	441:
		tmrA_10.PT := T#60S;
		tmrA_10.IN := TRUE;
		stepA := stepA + 1;
			 
	442:// 到達中間感應器，停止
		IF NOT io.i202 OR tmrA_10.q THEN
			io.q201 := FALSE;
			tmrA_10.in := FALSE;
					  
			IF NOT io.i202 THEN
				stepA := stepA + 1;
			ELSIF tmrA_10.q THEN
				stepA := stepA + 10000;
			END_IF
		END_IF
			 
	443:
		tmrA_1.PT := T#500ms;
		tmrA_1.IN := TRUE;
		IF tmrA_1.Q THEN
			tmrA_1.IN := FALSE;
			io.q202 := TRUE;
			IF io.i202 THEN
				// 如果上升到超過感應器，下降到有之後，繼續下降到脫離
				stepA := 444;
			ELSE
				// 停在感應器上，下降到脫離
				stepA := 445;
			END_IF
		END_IF
			
	444:// 
		IF NOT io.i202 THEN
			stepA := stepA + 1;
		END_IF
				  
	445:
		IF io.i202 THEN
			io.q202 := FALSE;
			stepA := stepA + 1;
		END_IF
				  
	446:
		CarLift_WaitSync.0 := TRUE;
		stepA := 450;
				  
//	450: // 等待主油壓切至慢速模式 ，完成後由主流程跳步
				  
	451: // 用慢速上升
		io.q201 := TRUE;
		IF NOT io.i202 THEN
			io.q201 := FALSE;
			stepA := stepA + 1;
		END_IF
				  
	452: // 用慢速上升
		io.q201 := TRUE;
		IF NOT io.i202 THEN
			io.q201 := FALSE;
			stepA := stepA + 1;
		END_IF
		
	453:
		stepA := 0;
	{endregion}
			  
	{region "============= 位置不確定  ============="}	
	470: // 位置不確定(沒在任何感應器上) ，先下降
		io.q201 := FALSE;
		io.q202 := TRUE;
		stepA := stepA + 1;
			 
	471:
		tmrA_10.PT := T#60S;
		tmrA_10.IN := TRUE;
		stepA := stepA + 1;
			 
	472:// 通過中間感應器 或 到達下方感應器
		IF NOT io.i202 OR NOT io.i203 OR tmrA_10.q THEN
			tmrA_10.in := FALSE;
					  
			IF NOT io.i203 THEN
				// 到達下方感應器
				io.q202 := FALSE;
				stepA := 440;
			ELSIF NOT io.i202 THEN
				// 通過中間感應器
				stepA := 480;
			ELSIF tmrA_10.q THEN
				stepA := stepA + 10000;
			END_IF
		END_IF
			 
	480: 
		IF io.i202 THEN
			io.q202 := FALSE;
			stepA := stepA + 1;
		END_IF
			
	481:// 
		CarLift_WaitSync.0 := TRUE;
		stepA := 420;
	{endregion}
		
END_CASE
{endregion}

{region "============= 台車B中位移動  ============="}
CASE stepB OF
	400: // 判斷位置
		IF NOT io.i205 THEN
			stepB := 0;
		ELSE
			IF NOT io.i204 THEN
				// 位置在上限
				stepB := 410;
			ELSIF NOT io.i206 THEN
				// 位置在下限
				stepB := 440;
			ELSE
			    // 位置不確定
				stepB := 470;
		 	END_IF
		END_IF
	{region "============= 位置在上限  ============="}	
	410: // 位置在上限，下降
		io.q203 := FALSE;
		io.q204 := TRUE;
		stepB := stepB + 1;
			 
	411:
		tmrB_10.PT := T#60S;
		tmrB_10.IN := TRUE;
		stepB := stepB + 1;
			 
	412://
		IF NOT io.i205 OR tmrB_10.q THEN
			tmrB_10.in := FALSE;
			IF NOT io.i205 THEN
				stepB := stepB + 1;
			ELSIF tmrB_10.q THEN
				stepB := stepB + 10000;
			END_IF
		END_IF
			 
	413: // 先降過頭在慢速升回
		IF io.i205 THEN
			io.q204 := FALSE;
			stepB := stepB + 1;
		END_IF
				  
	414:
		CarLift_WaitSync.1 := TRUE;
		stepB := 420;
				  
//	420: // 等待主油壓切至慢速模式 ，完成後由主流程跳步
		
				  
	421: // 用慢速上升
		io.q203 := TRUE;
		IF NOT io.i205 THEN
			io.q203 := FALSE;
			stepB := stepB + 1;
		END_IF
				  
	422: // 用慢速上升
		io.q203 := TRUE;
		IF NOT io.i205 THEN
			io.q203 := FALSE;
			stepB := stepB + 1;
		END_IF
		
	423:
		stepB := 0;
	{endregion}
	{region "============= 位置在下限  ============="}	
	440: // 位置在下限，上升
		io.q203 := TRUE;
		io.q204 := FALSE;
		stepB := stepB + 1;
			 
	441:
		tmrB_10.PT := T#60S;
		tmrB_10.IN := TRUE;
		stepB := stepB + 1;
			 
	442:// 到達中間感應器，停止
		IF NOT io.i205 OR tmrB_10.q THEN
			io.q203 := FALSE;
			tmrB_10.in := FALSE;
					  
			IF NOT io.i205 THEN
				stepB := stepB + 1;
			ELSIF tmrB_10.q THEN
				stepB := stepB + 10000;
			END_IF
		END_IF
			 
	443:
		tmrB_1.PT := T#500ms;
		tmrB_1.IN := TRUE;
		IF tmrB_1.Q THEN
			tmrB_1.IN := FALSE;
			io.q204 := TRUE;
			IF io.i205 THEN
				// 如果上升到超過感應器，下降到有之後，繼續下降到脫離
				stepB := 444;
			ELSE
				// 停在感應器上，下降到脫離
				stepB := 445;
			END_IF
		END_IF
			
	444:// 
		IF NOT io.i205 THEN
			stepB := stepB + 1;
		END_IF
				  
	445:
		IF io.i205 THEN
			io.q204 := FALSE;
			stepB := stepB + 1;
		END_IF
				  
	446:
		CarLift_WaitSync.1 := TRUE;
		stepB := 450;
				  
//	450: // 等待主油壓切至慢速模式 ，完成後由主流程跳步
				  
	451: // 用慢速上升
		io.q203 := TRUE;
		IF NOT io.i205 THEN
			io.q203 := FALSE;
			stepB := stepB + 1;
		END_IF
				  
	452: // 用慢速上升
		io.q203 := TRUE;
		IF NOT io.i205 THEN
			io.q203 := FALSE;
			stepB := stepB + 1;
		END_IF
		
	453:
		stepB := 0;
	{endregion}
			  
	{region "============= 位置不確定  ============="}	
	470: // 位置不確定(沒在任何感應器上) ，先下降
		io.q203 := FALSE;
		io.q204 := TRUE;
		stepB := stepB + 1;
			 
	471:
		tmrB_10.PT := T#60S;
		tmrB_10.IN := TRUE;
		stepB := stepB + 1;
			 
	472:// 通過中間感應器 或 到達下方感應器
		IF NOT io.i205 OR NOT io.i206 OR tmrB_10.q THEN
			tmrB_10.in := FALSE;
					  
			IF NOT io.i206 THEN
				// 到達下方感應器
				io.q204 := FALSE;
				stepB := 440;
			ELSIF NOT io.i205 THEN
				// 通過中間感應器
				stepB := 480;
			ELSIF tmrB_10.q THEN
				stepB := stepB + 10000;
			END_IF
		END_IF
			 
	480: 
		IF io.i205 THEN
			io.q204 := FALSE;
			stepB := stepB + 1;
		END_IF
			
	481:// 
		CarLift_WaitSync.1 := TRUE;
		stepB := 420;
	{endregion}
		
END_CASE
{endregion}
	 
{region "============= 台車C中位移動  ============="}
CASE stepC OF
	400: // 判斷位置
		IF NOT io.i208 THEN
			stepC := 0;
		ELSE
			IF NOT io.i207 THEN
				// 位置在上限
				stepC := 410;
			ELSIF NOT io.i209 THEN
				// 位置在下限
				stepC := 440;
			ELSE
			    // 位置不確定
				stepC := 470;
		 	END_IF
		END_IF
	{region "============= 位置在上限  ============="}	
	410: // 位置在上限，下降
		io.q205 := FALSE;
		io.q206 := TRUE;
		stepC := stepC + 1;
			 
	411:
		tmrC_10.PT := T#60S;
		tmrC_10.IN := TRUE;
		stepC := stepC + 1;
			 
	412://
		IF NOT io.i208 OR tmrC_10.q THEN
			tmrC_10.in := FALSE;
			IF NOT io.i208 THEN
				stepC := stepC + 1;
			ELSIF tmrC_10.q THEN
				stepC := stepC + 10000;
			END_IF
		END_IF
			 
	413: // 先降過頭在慢速升回
		IF io.i208 THEN
			io.q206 := FALSE;
			stepC := stepC + 1;
		END_IF
				  
	414:
		CarLift_WaitSync.2 := TRUE;
		stepC := 420;
				  
//	420: // 等待主油壓切至慢速模式 ，完成後由主流程跳步
		
				  
	421: // 用慢速上升
		io.q205 := TRUE;
		IF NOT io.i208 THEN
			io.q205 := FALSE;
			stepC := stepC + 1;
		END_IF
				  
	422: // 用慢速上升
		io.q205 := TRUE;
		IF NOT io.i208 THEN
			io.q205 := FALSE;
			stepC := stepC + 1;
		END_IF
		
	423:
		stepC := 0;
	{endregion}
	{region "============= 位置在下限  ============="}	
	440: // 位置在下限，上升
		io.q205 := TRUE;
		io.q206 := FALSE;
		stepC := stepC + 1;
			 
	441:
		tmrC_10.PT := T#60S;
		tmrC_10.IN := TRUE;
		stepC := stepC + 1;
			 
	442:// 到達中間感應器，停止
		IF NOT io.i208 OR tmrC_10.q THEN
			io.q205 := FALSE;
			tmrC_10.in := FALSE;
					  
			IF NOT io.i208 THEN
				stepC := stepC + 1;
			ELSIF tmrC_10.q THEN
				stepC := stepC + 10000;
			END_IF
		END_IF
			 
	443:
		tmrC_1.PT := T#500ms;
		tmrC_1.IN := TRUE;
		IF tmrC_1.Q THEN
			tmrC_1.IN := FALSE;
			io.q206 := TRUE;
			IF io.i208 THEN
				// 如果上升到超過感應器，下降到有之後，繼續下降到脫離
				stepC := 444;
			ELSE
				// 停在感應器上，下降到脫離
				stepC := 445;
			END_IF
		END_IF
			
	444:// 
		IF NOT io.i208 THEN
			stepC := stepC + 1;
		END_IF
				  
	445:
		IF io.i208 THEN
			io.q206 := FALSE;
			stepC := stepC + 1;
		END_IF
				  
	446:
		CarLift_WaitSync.2 := TRUE;
		stepC := 450;
				  
//	450: // 等待主油壓切至慢速模式 ，完成後由主流程跳步
				  
	451: // 用慢速上升
		io.q205 := TRUE;
		IF NOT io.i208 THEN
			io.q205 := FALSE;
			stepC := stepC + 1;
		END_IF
				  
	452: // 用慢速上升
		io.q205 := TRUE;
		IF NOT io.i208 THEN
			io.q205 := FALSE;
			stepC := stepC + 1;
		END_IF
		
	453:
		stepC := 0;
	{endregion}
			  
	{region "============= 位置不確定  ============="}	
	470: // 位置不確定(沒在任何感應器上) ，先下降
		io.q205 := FALSE;
		io.q206 := TRUE;
		stepC := stepC + 1;
			 
	471:
		tmrC_10.PT := T#60S;
		tmrC_10.IN := TRUE;
		stepC := stepC + 1;
			 
	472:// 通過中間感應器 或 到達下方感應器
		IF NOT io.i208 OR NOT io.i209 OR tmrC_10.q THEN
			tmrC_10.in := FALSE;
					  
			IF NOT io.i209 THEN
				// 到達下方感應器
				io.q206 := FALSE;
				stepC := 440;
			ELSIF NOT io.i208 THEN
				// 通過中間感應器
				stepC := 480;
			ELSIF tmrC_10.q THEN
				stepC := stepC + 10000;
			END_IF
		END_IF
			 
	480: 
		IF io.i208 THEN
			io.q206 := FALSE;
			stepC := stepC + 1;
		END_IF
			
	481:// 
		CarLift_WaitSync.2 := TRUE;
		stepC := 420;
	{endregion}
		
END_CASE
{endregion}
	 
{region "============= 台車D中位移動  ============="}
CASE stepD OF
	400: // 判斷位置
		IF NOT io.i211 THEN
			stepD := 0;
		ELSE
			IF NOT io.i210 THEN
				// 位置在上限
				stepD := 410;
			ELSIF NOT io.i212 THEN
				// 位置在下限
				stepD := 440;
			ELSE
			    // 位置不確定
				stepD := 470;
		 	END_IF
		END_IF
	{region "============= 位置在上限  ============="}	
	410: // 位置在上限，下降
		io.q207 := FALSE;
		io.q208 := TRUE;
		stepD := stepD + 1;
			 
	411:
		tmrD_10.PT := T#60S;
		tmrD_10.IN := TRUE;
		stepD := stepD + 1;
			 
	412://
		IF NOT io.i211 OR tmrD_10.q THEN
			tmrD_10.in := FALSE;
			IF NOT io.i211 THEN
				stepD := stepD + 1;
			ELSIF tmrD_10.q THEN
				stepD := stepD + 10000;
			END_IF
		END_IF
			 
	413: // 先降過頭在慢速升回
		IF io.i211 THEN
			io.q208 := FALSE;
			stepD := stepD + 1;
		END_IF
				  
	414:
		CarLift_WaitSync.3 := TRUE;
		stepD := 420;
				  
//	420: // 等待主油壓切至慢速模式 ，完成後由主流程跳步
		
				  
	421: // 用慢速上升
		io.q207 := TRUE;
		IF NOT io.i211 THEN
			io.q207 := FALSE;
			stepD := stepD + 1;
		END_IF
				  
	422: // 用慢速上升
		io.q207 := TRUE;
		IF NOT io.i211 THEN
			io.q207 := FALSE;
			stepD := stepD + 1;
		END_IF
		
	423:
		stepD := 0;
	{endregion}
	{region "============= 位置在下限  ============="}	
	440: // 位置在下限，上升
		io.q207 := TRUE;
		io.q208 := FALSE;
		stepD := stepD + 1;
			 
	441:
		tmrD_10.PT := T#60S;
		tmrD_10.IN := TRUE;
		stepD := stepD + 1;
			 
	442:// 到達中間感應器，停止
		IF NOT io.i211 OR tmrD_10.q THEN
			io.q207 := FALSE;
			tmrD_10.in := FALSE;
					  
			IF NOT io.i211 THEN
				stepD := stepD + 1;
			ELSIF tmrD_10.q THEN
				stepD := stepD + 10000;
			END_IF
		END_IF
			 
	443:
		tmrD_1.PT := T#500ms;
		tmrD_1.IN := TRUE;
		IF tmrD_1.Q THEN
			tmrD_1.IN := FALSE;
			io.q208 := TRUE;
			IF io.i211 THEN
				// 如果上升到超過感應器，下降到有之後，繼續下降到脫離
				stepD := 444;
			ELSE
				// 停在感應器上，下降到脫離
				stepD := 445;
			END_IF
		END_IF
			
	444:// 
		IF NOT io.i211 THEN
			stepD := stepD + 1;
		END_IF
				  
	445:
		IF io.i211 THEN
			io.q208 := FALSE;
			stepD := stepD + 1;
		END_IF
				  
	446:
		CarLift_WaitSync.3 := TRUE;
		stepD := 450;
				  
//	450: // 等待主油壓切至慢速模式 ，完成後由主流程跳步
				  
	451: // 用慢速上升
		io.q207 := TRUE;
		IF NOT io.i211 THEN
			io.q207 := FALSE;
			stepD := stepD + 1;
		END_IF
				  
	452: // 用慢速上升
		io.q207 := TRUE;
		IF NOT io.i211 THEN
			io.q207 := FALSE;
			stepD := stepD + 1;
		END_IF
		
	453:
		stepD := 0;
	{endregion}
			  
	{region "============= 位置不確定  ============="}	
	470: // 位置不確定(沒在任何感應器上) ，先下降
		io.q207 := FALSE;
		io.q208 := TRUE;
		stepD := stepD + 1;
			 
	471:
		tmrD_10.PT := T#60S;
		tmrD_10.IN := TRUE;
		stepD := stepD + 1;
			 
	472:// 通過中間感應器 或 到達下方感應器
		IF NOT io.i211 OR NOT io.i212 OR tmrD_10.q THEN
			tmrD_10.in := FALSE;
					  
			IF NOT io.i212 THEN
				// 到達下方感應器
				io.q208 := FALSE;
				stepD := 440;
			ELSIF NOT io.i211 THEN
				// 通過中間感應器
				stepD := 480;
			ELSIF tmrD_10.q THEN
				stepD := stepD + 10000;
			END_IF
		END_IF
			 
	480: 
		IF io.i211 THEN
			io.q208 := FALSE;
			stepD := stepD + 1;
		END_IF
			
	481:// 
		CarLift_WaitSync.3 := TRUE;
		stepD := 420;
	{endregion}
		
END_CASE
{endregion}
END_ACTION

ACTION step_6_CarLift_Down:
CASE step OF
	600:
		IF (CarLift_Select AND 16#F) = 0 THEN
			CarLift_Select := 15;
		END_IF
		step := step + 1;
	
	601:
		io.q301 := TRUE;
		IF CarLift_Select.0 THEN
			stepA := 600;
		END_IF
		
		IF CarLift_Select.1 THEN
			stepB := 600;
		END_IF
		
		IF CarLift_Select.2 THEN
			stepC := 600;
		END_IF
		
		IF CarLift_Select.3 THEN
			stepD := 600;
		END_IF
		
		step := step + 1;
		
	602:
		IF stepA = 0 AND stepB = 0 AND stepC = 0 AND stepD = 0 THEN
			step := step + 1;
		ELSIF stepA > 10000 OR stepB > 10000 OR stepC > 10000 OR stepD > 10000 THEN
			step := step + 10000;
		END_IF
		
	603:
		io.q301 := FALSE;
		CarLift_Select := 0;
		bDone := TRUE;
		step := 0;
		
END_CASE

{region "============= 台車A下降  ============="}
CASE stepA OF
	600: // 啟動上升
		io.q201 := FALSE;
		io.q202 := TRUE;
		stepA := stepA + 1;
		
	601: // 啟動超時計時器
		tmrA_10.PT := T#20S;
		tmrA_10.IN := TRUE;
		stepA := stepA + 1;
		
	602: // 等待
		IF NOT io.i203 OR tmrA_10.q THEN
			tmrA_10.in := FALSE;
			
			IF NOT io.i203 THEN
				stepA := stepA + 1;
			ELSIF tmrA_10.q THEN
				io.q202 := FALSE;
				stepA := stepA + 10000;
			END_IF
		END_IF
		
	603: // 成功之後等待1秒
		tmrA_1.PT := T#1S;
		tmrA_1.IN := TRUE;
		IF tmrA_1.Q THEN
			tmrA_1.IN := FALSE;
			io.q202 := FALSE;
			stepA := stepA + 1;
		END_IF
		
	604:
		stepA := 0;
		
END_CASE
{endregion}

{region "============= 台車B下降  ============="}
CASE stepB OF
	600: // 啟動上升
		io.q203 := FALSE;
		io.q204 := TRUE;
		stepB := stepB + 1;
		
	601: // 啟動超時計時器
		tmrB_10.PT := T#20S;
		tmrB_10.IN := TRUE;
		stepB := stepB + 1;
		
	602: // 等待
		IF NOT io.i206 OR tmrB_10.q THEN
			tmrB_10.in := FALSE;
			
			IF NOT io.i206 THEN
				stepB := stepB + 1;
			ELSIF tmrB_10.q THEN
				io.q204 := FALSE;
				stepB := stepB + 10000;
			END_IF
		END_IF
		
	603: // 成功之後等待1秒
		tmrB_1.PT := T#1S;
		tmrB_1.IN := TRUE;
		IF tmrB_1.Q THEN
			io.q204 := FALSE;
			stepB := stepB + 1;
		END_IF
		
	604:
		stepB := 0;
		
END_CASE
{endregion}

{region "============= 台車C下降  ============="}
CASE stepC OF
	600: // 啟動上升
		io.q205 := FALSE;
		io.q206 := TRUE;
		stepC := stepC + 1;
		
	601: // 啟動超時計時器
		tmrC_10.PT := T#20S;
		tmrC_10.IN := TRUE;
		stepC := stepC + 1;
		
	602: // 等待
		IF NOT io.i209 OR tmrC_10.q THEN
			tmrC_10.in := FALSE;
			
			IF NOT io.i209 THEN
				stepC := stepC + 1;
			ELSIF tmrC_10.q THEN
				io.q206 := FALSE;
				stepC := stepC + 10000;
			END_IF
		END_IF
		
	603: // 成功之後等待1秒
		tmrC_1.PT := T#1S;
		tmrC_1.IN := TRUE;
		IF tmrC_1.Q THEN
			io.q206 := FALSE;
			stepC := stepC + 1;
		END_IF
		
	604:
		stepC := 0;
		
END_CASE
{endregion}

{region "============= 台車D下降  ============="}
CASE stepD OF
	600: // 啟動上升
		io.q207 := FALSE;
		io.q208 := TRUE;
		stepD := stepD + 1;
		
	601: // 啟動超時計時器
		tmrD_10.PT := T#20S;
		tmrD_10.IN := TRUE;
		stepD := stepD + 1;
		
	602: // 等待
		IF NOT io.i212 OR tmrD_10.q THEN
			tmrD_10.in := FALSE;
			
			IF NOT io.i212 THEN
				stepD := stepD + 1;
			ELSIF tmrD_10.q THEN
				io.q207 := FALSE;
				stepD := stepD + 10000;
			END_IF
		END_IF
		
	603: // 成功之後等待1秒
		tmrD_1.PT := T#1S;
		tmrD_1.IN := TRUE;
		IF tmrD_1.Q THEN
			io.q208 := FALSE;
			stepD := stepD + 1;
		END_IF
		
	604:
		stepD := 0;
		
END_CASE
{endregion}
END_ACTION

ACTION step1_1_Pull_over:
CASE step1 OF
	100:// 檢查
		TryCount := 0;
		step1 := step1 + 1;
		
	101:
		step1 := 110;
		
	110: // 啟動靠邊油壓閥
		io.q302 := TRUE;
		IF NOT bbuzy THEN
			io.q301 := TRUE;
		END_IF
		step1 := step1 + 1;
		
	111: // 確定原點已脫離
		IF io.i401 THEN
			step1 := step1 + 1;
		END_IF
		
	112: // 程序暫停5秒
		tmr1_01.PT := T#4S;
		tmr1_01.IN := io.i402 OR io.i404;
		
		tmr1_02.PT := T#5S;
		tmr1_02.IN := TRUE;
		IF tmr1_01.Q OR tmr1_02.q THEN
			tmr1_01.IN := FALSE;
			tmr1_02.IN := FALSE;
			
			IF tmr1_01.q THEN
				step1 := 190;
			ELSIF tmr1_02.Q THEN
				step1 := step1 + 1;
			END_IF
		END_IF
		
	113:
		step1 := 120;
		
	120:// 沒推到待命位置
		io.q302 := FALSE;
		step1 := step1 + 1;
		
	121: // 等待回原點
		tmr01.PT := T#1S;
		tmr01.IN := (NOT io.i401 AND NOT io.i403 AND NOT io.i405 AND NOT io.i407);
		IF tmr01.Q THEN
			tmr01.IN := FALSE;
			step1 := step1 + 1;
		END_IF
		
	122: 
		
		IF TryCount < 4 THEN
			TryCount := TryCount + 1;
			step1 := 110;
		ELSE
			TryCount := 0;
			step1 := step1 + 10000;
		END_IF
		
		
	190:
		
		tmr1_01.PT := T#3S;
		tmr1_01.IN := TRUE;
		IF tmr1_01.Q THEN
			tmr1_01.IN := FALSE;
			step1 := step1 + 1;
		END_IF
		
	191:
		io.q302 := FALSE;
		bdone1 := TRUE;
		step1 := 0;
END_CASE
END_ACTION

ACTION step1_2_Pull_over_Jog:
CASE step1 OF
	200:// 檢查
		step1 := step1 + 1;
		
	201:
		IF io.q302 THEN
			step1 := 220;
		ELSE
			step1 := 210;
		END_IF
		
		
	210: // 啟動靠邊油壓閥
		io.q302 := TRUE;
		IF NOT bbuzy THEN
			io.q301 := TRUE;
		END_IF
		step1 := step1 + 1;
		
	211: // 確定原點已脫離
		tmr01.PT := T#4S;
		tmr01.IN := (io.i401 AND io.i403 AND io.i405 AND io.i407);
		IF tmr01.Q THEN
			tmr01.IN := FALSE;
			step1 := step1 + 1;
		END_IF
		
	212:
		step1 := 290;
		
	220: // 關閉靠邊油壓閥
		io.q302 := FALSE;
		IF NOT bbuzy THEN
			io.q301 := TRUE;
		END_IF
		step1 := step1 + 1;
		
	221: // 等待回原點
		tmr01.PT := T#4S;
		tmr01.IN := (NOT io.i401 AND NOT io.i403 AND NOT io.i405 AND NOT io.i407);
		IF tmr01.Q THEN
			tmr01.IN := FALSE;
			step1 := step1 + 1;
		END_IF
		
	222: 
		step1 := 290;
		
		
	290:
		bdone1 := TRUE;
		io.q301 := FALSE;
		step1 := 0;
END_CASE
END_ACTION

METHOD Stop : BOOL
VAR_INPUT
END_VAR
step := 100;
END_METHOD

ACTION tmrAct:
tmr01();

tmr1_01();
tmr1_02();

tmrA_1();
tmrA_10();
tmrB_1();
tmrB_10();
tmrC_1();
tmrC_10();
tmrD_1();
tmrD_10();


tmr_pump();
END_ACTION

END_PROGRAM

// ---- POUs/動作流程控制/滾輪整料/PullOver.TcPOU
PROGRAM PullOver
VAR
	step: UINT;
	
	
END_VAR

VAR_OUTPUT
	bBuzy: BOOL;
	bError: BOOL;
	bDone: BOOL;
	iErrorId : DINT;
END_VAR

IF (EStop OR SystemError OR Input.Feed_Reset) AND bBuzy THEN
	IF bBuzy THEN
		step := step  + 10000;
	END_IF
END_IF

bBuzy := (step >= 1 AND step < 10000);
bError := (step > 10000);


CASE step OF
	1:
		bDone := FALSE;
		step := 10;	
(*	=====================================
				測高不再原點
	=====================================*)
	10:
		IF HeightMeasurer.at_Home THEN
			step := 100;
		ELSE
			step := step + 1;
		END_IF
		
	11:
		HeightMeasurer.Homing();
		step := step + 1;
		
	12:
		IF HeightMeasurer.bBuzy OR HeightMeasurer.bError THEN
			step := step + 1;
		END_IF
		
	13:
		IF HeightMeasurer.bDone THEN
			step := step + 1;
		ELSIF HeightMeasurer.bError THEN
			step := step + 10000;
		END_IF
		
	14:
		step := 100;
		
		
(*	=====================================
				靠邊啟動
	=====================================*)
	100:
		Hydraulic.Over_Pull(0);
		step := step + 1;
		
	101:
		IF (Hydraulic.bBuzy1 OR Hydraulic.bError1) THEN
			step := step + 1;
		END_IF
		
	102:
		IF Hydraulic.bDone1 THEN
			step := step + 1;
		ELSIF Hydraulic.bError1 THEN
			step := step + 10000;
		END_IF
		
	103:
		step := 110;
		
(*	=====================================
				高度測量
	=====================================*)
	110:
		HeightMeasurer.Measure();
		step := step + 1;
		
	111:
		IF (HeightMeasurer.bBuzy OR HeightMeasurer.bError) THEN
			step := step + 1;
		END_IF
		
	112:
		IF HeightMeasurer.bDone THEN
			step := step + 1;
		ELSIF HeightMeasurer.bError THEN
			step := step + 10000;
		END_IF
		
	113:
		step := 120;
		
	
	120:
		bDone := TRUE;
		step := 0;
END_CASE

IF Input.PullOver_Start AND NOT bBuzy THEN
	step := 1;
END_IF

Output.PullOver_bBuzy := bBuzy;
Output.PullOver_bDone := bDone;
Output.PullOver_bError := bError;

METHOD Start
VAR_INPUT
END_VAR
step := 1;
END_METHOD

END_PROGRAM

// ---- POUs/硬體控制/進料滾輪/FeedRoller.TcPOU
PROGRAM FeedRoller
VAR
	step: INT;
	
	_run : BOOL;
	
	start_RTrig : R_TRIG;
	start_FTrig : F_TRIG;
	
	_bError : BOOL;
	
	tmr0 : TON;
	tmr1 : TON;
END_VAR

VAR_OUTPUT
	bDone: BOOL;
	bBuzy: BOOL;
	bError: BOOL;
	
	Move_Fwd : BOOL;
	Move_Rev : BOOL;
	At_Up : BOOL;
	At_Down : BOOL;
END_VAR

// 沒 SystemError 是避免進料機影響到整體動作
IF (EStop OR Input.Feed_Reset) AND bBuzy THEN
	IF bBuzy THEN
		step := step  + 10000;
	END_IF
	IO.q102 := FALSE;
	IO.q103 := FALSE;
	IO.q309 := FALSE;
	IO.q310 := FALSE;
	IO.q311 := FALSE;
	IO.q312 := FALSE;
END_IF


// 外部 送入 啟動訊號
start_RTrig(CLK := Input.In_Moter_Start );

IF	start_RTrig.q THEN
	step := 1;
END_IF

// 外部 解除 啟動訊號
start_FTrig(CLK := Input.In_Moter_Start);

IF start_FTrig.Q THEN
	step := 100;
END_IF

// 執行動作發生錯誤
_bError := step > 10000;

IF _bError THEN
	_run := FALSE;
	IO.q103 := FALSE;
	IO.q102 := FALSE;
END_IF

// 馬達 動作中過載檢知
IF IO.i109 AND step > 0 AND step < 10000 THEN
	step := 10900;
END_IF

bBuzy := step > 0 AND step < 10000;
bError := step > 10000;

IF bBuzy THEN
	bDone := FALSE;
END_IF

step_0_Auto_Start();
step_1_Auto_Stop();
step_7_Jog_FwdRev();
step_8_Jog_UpDown();

Output.In_Moter_Running := step > 0 OR Move_Fwd OR Move_Rev;
Output.In_Moter_Error := _bError;

tmr0();
tmr1();

Move_Fwd	:= IO.q103;
Move_Rev	:= IO.q102;
At_Up		:= IO.i411;
At_Down		:= IO.i412;

METHOD Jog_Down
VAR_INPUT
END_VAR
bDone := FALSE;

step := 820;
END_METHOD

METHOD Jog_Fwd
VAR_INPUT
END_VAR
bDone := FALSE;

step := 700;
END_METHOD

METHOD Jog_Rev
VAR_INPUT
END_VAR
bDone := FALSE;

step := 720;
END_METHOD

METHOD Jog_Stop
VAR_INPUT
END_VAR
step := 780;
END_METHOD

METHOD Jog_Up
VAR_INPUT
END_VAR
bDone := FALSE;

step := 800;
END_METHOD

ACTION step_0_Auto_Start:
CASE step OF
	1:
		IF IO.i109 THEN
			// 滾輪馬達保護氣跳脫
			step := step + 10000;
// 		ELSIF NOT IO.i314 THEN
// 			// 測高位置錯誤
// 			step := step + 10000;
		ELSE
			step := step + 1;
		END_IF
		
	2:
		IF HeightMeasurer.bBuzy THEN
			// 測高動作執行中
			step := step + 10000;
		ELSE
			// 進料動作執行中
			step := step + 1;
		END_IF
		
	3:
		step := 10;
		
	10:
		IO.q309 := TRUE;
		IO.q310 := FALSE;
		IO.q311 := TRUE;
		IO.q312 := FALSE;
		tmr1.PT := T#10S;
		tmr1.IN := TRUE;
		step := step + 1;
		
	11:
		IF NOT IO.i412 OR tmr1.Q THEN
			IO.q309 := FALSE;
			IO.q311 := FALSE;
			tmr1.IN := FALSE;
			IF NOT IO.i412 THEN
				step := step + 1;
			ELSE
				// 上升超時
				step := step + 10000;
			END_IF
		END_IF
		
	12:
		step := 20;
		
	20:
		IO.q103 := TRUE;
		_run :=	TRUE;
		step := 0;
END_CASE
END_ACTION

ACTION step_1_Auto_Stop:
CASE step OF
	100:
		IO.q309 := FALSE;
		IO.q311 := FALSE;
		IO.q103 := FALSE;
		step := step + 1;
		
	101:
		tmr0.PT:= T#1S;
		tmr0.IN := TRUE;
		IF tmr0.Q THEN
			tmr0.IN := FALSE;
			step := step + 1;
		END_IF
		
	102:
		step := 110;
		
	110:
		IO.q310 := TRUE;
		IO.q312 := TRUE;
		tmr1.PT := T#10S;
		tmr1.IN := TRUE;
		step := step + 1;
		
	111:
		IF IO.i412 OR tmr1.Q THEN
			IO.q310 := FALSE;
			IO.q312 := FALSE;
			tmr1.IN := FALSE;
			IF IO.i412 THEN
				step := step + 1;
			ELSE
				// 上升超時
				step := step + 10000;
			END_IF
		END_IF
		
	112:
		_run :=	FALSE;
		step := 0;
END_CASE
END_ACTION

ACTION step_7_Jog_FwdRev:
CASE step OF
	700:
		IO.q102 := FALSE;
		IF IO.i109 THEN
			// 滾輪馬達保護氣跳脫
			step := step + 10000;
// 		ELSIF NOT IO.i314 THEN
// 			// 測高位置錯誤
// 			step := step + 10000;
		ELSE
			step := step + 1;
		END_IF
		
	701: // 啟動馬達
		IO.q103 := TRUE;
		bDone := TRUE;
		step := 0;
		
	
		


	720:
		IO.q103 := FALSE;
		IF IO.i109 THEN
			// 滾輪馬達保護氣跳脫
			step := step + 10000;
// 		ELSIF NOT IO.i314 THEN
// 			// 測高位置錯誤
// 			step := step + 10000;
		ELSE
			step := step + 1;
		END_IF
		
	721:
		IO.q102 := TRUE;
		bDone := TRUE;
		step := 0;
		
	
		


	780:
		IO.q102 := FALSE;
		IO.q103 := FALSE;
		bDone := TRUE;
		step := 0;
END_CASE
END_ACTION

ACTION step_8_Jog_UpDown:
CASE step OF
	800:
		IO.q309 := TRUE;
		IO.q310 := FALSE;
		IO.q311 := TRUE;
		IO.q312 := FALSE;
		
		tmr1.PT := T#10S;
		tmr1.IN := TRUE;
		step := step + 1;
		
	801: // 滾輪上升
		IF NOT IO.i412 OR tmr1.Q THEN
			IO.q309 := FALSE;
			IO.q311 := FALSE;
			tmr1.IN := FALSE;
			IF NOT IO.i412 THEN
				step := step + 1;
			ELSE
				// 上升超時
				step := step + 10000;
			END_IF
		END_IF
		
	802:
		bDone := TRUE;
		step := 0;
		
	
		


	820:
		IO.q309 := FALSE;
		IO.q310 := TRUE;
		IO.q311 := FALSE;
		IO.q312 := TRUE;
		
		tmr1.PT := T#10S;
		tmr1.IN := TRUE;
		step := step + 1;
		
	821: // 滾輪上升
		IF IO.i412 OR tmr1.Q THEN
			IO.q310 := FALSE;
			IO.q312 := FALSE;
			tmr1.IN := FALSE;
			IF IO.i412 THEN
				step := step + 1;
			ELSE
				// 上升超時
				step := step + 10000;
			END_IF
		END_IF
		
	822:
		bDone := TRUE;
		step := 0;
		
	

END_CASE
END_ACTION

END_PROGRAM

// ---- POUs/硬體控制/出料滾輪/ProductRoller.TcPOU
PROGRAM ProductRoller
VAR
	step: INT;
	
	_run : BOOL;
	
	start_RTrig : R_TRIG;
	start_FTrig : F_TRIG;
	
	_bError : BOOL;
	
	
	tmr0 : TON;
	tmr1 : TON;
	
	Roller_Up :BOOL;
	Roller_Down :BOOL;
	
	Roller_Fwd :BOOL;
	Roller_Rev :BOOL;
END_VAR

VAR_OUTPUT
	bDone: BOOL;
	bBuzy: BOOL;
	bError: BOOL;
	
	Move_Fwd : BOOL;
	Move_Rev : BOOL;
	At_Up : BOOL;
	At_Down : BOOL;
END_VAR


// 沒 SystemError 是避免進料機影響到整體動作
IF (EStop OR Input.Feed_Reset) AND bBuzy THEN
	IF bBuzy THEN
		step := step  + 10000;
	END_IF
	IO.q114 := FALSE;
	IO.q115 := FALSE;
	IO.q305 := FALSE;
	IO.q306 := FALSE;
END_IF


// 外部 送入 啟動訊號
start_RTrig(CLK := Input.Out_Moter_Start);

IF	start_RTrig.q THEN
	step := 1;
END_IF

// 外部 解除 啟動訊號
start_FTrig(CLK := Input.Out_Moter_Start);

IF start_FTrig.Q THEN
	step := 100;
END_IF



// 執行動作發生錯誤
_bError := step > 10000;

IF _bError THEN
	_run := FALSE;
	IO.q114 := FALSE;
	IO.q115 := FALSE;
END_IF

// 馬達 動作中過載檢知
IF IO.i109 AND step > 0 AND step < 10000 THEN
	step := 10900;
END_IF

bBuzy := step > 0 AND step < 10000;
bError := step > 10000;

IF bBuzy THEN
	bDone := FALSE;
END_IF

IF NOT Pause THEN
	step_0_Auto_Start();
	step_1_Auto_Stop();

	IO.q115 := Roller_Fwd;
	IO.q114 := Roller_Rev;
	IO.q306 := Roller_Up;
	IO.q305 := Roller_Down;
ELSE
	IO.q115 := FALSE;
	IO.q114 := FALSE;
	IO.q306 := FALSE;
	IO.q305 := FALSE;
END_IF

step_7_Jog_FwdRev();
step_8_Jog_UpDown();



Output.Out_Moter_Running := step > 0 OR Move_Fwd OR Move_Rev;;
Output.Out_Moter_Error := _bError;

tmr0();
tmr1();

Move_Fwd	:= IO.q115;
Move_Rev	:= IO.q114;
At_Up		:= IO.i316;
At_Down		:= IO.i315;

METHOD Jog_Down
VAR_INPUT
END_VAR
bDone := FALSE;

step := 820;
END_METHOD

METHOD Jog_Fwd
VAR_INPUT
END_VAR
bDone := FALSE;

step := 700;
END_METHOD

METHOD Jog_Rev
VAR_INPUT
END_VAR
bDone := FALSE;

step := 720;
END_METHOD

METHOD Jog_Stop
VAR_INPUT
END_VAR
step := 780;
END_METHOD

METHOD Jog_Up
VAR_INPUT
END_VAR
bDone := FALSE;

step := 800;
END_METHOD

ACTION step_0_Auto_Start:
CASE step OF
	1:
		IF IO.i112 THEN
			// 滾輪馬達保護氣跳脫
			step := step + 10000;
// 		ELSIF IO.i113 THEN
// 			
		ELSE
			step := step + 1;
		END_IF
		
	2:
		step := 10;
		
	10:
		Roller_Down := FALSE;
		Roller_Up 	:= TRUE;
		tmr1.PT := T#10S;
		tmr1.IN := TRUE;
		step := step + 1;
		
	11:
		IF NOT IO.i315 OR tmr1.Q THEN
			Roller_Up := FALSE;
			tmr1.IN := FALSE;
			IF NOT IO.i315 THEN
				step := step + 1;
			ELSE
				// 上升超時
				step := step + 10000;
			END_IF
		END_IF
		
	12:
		step := 20;
		
	20:
		Roller_Rev := FALSE;
		Roller_Fwd := TRUE;
		_run :=	TRUE;
		step := 0;
END_CASE
END_ACTION

ACTION step_1_Auto_Stop:
CASE step OF
	100:
		Roller_Rev := FALSE;
		Roller_Fwd := FALSE;
		step := step + 1;
		
	101:
		tmr0.PT:= T#1S;
		tmr0.IN := TRUE;
		IF tmr0.Q THEN
			tmr0.IN := FALSE;
			step := step + 1;
		END_IF
		
	102:
		step := 110;
		
	110:
		Roller_Down := TRUE;
		Roller_Up := FALSE;
		tmr1.PT := T#10S;
		tmr1.IN := TRUE;
		step := step + 1;
		
	111:
		IF IO.i315 OR tmr1.Q THEN
			Roller_Down := FALSE;
			tmr1.IN := FALSE;
			IF IO.i315 THEN
				step := step + 1;
			ELSE
				// 上升超時
				step := step + 10000;
			END_IF
		END_IF
		
	112:
		_run :=	FALSE;
		step := 0;
END_CASE
END_ACTION

ACTION step_7_Jog_FwdRev:
CASE step OF
	700:
		Roller_Rev := FALSE;
		IF IO.i112 THEN
			// 滾輪馬達保護氣跳脫
			step := step + 10000;
		ELSE
			step := step + 1;
		END_IF
		
	701: // 啟動馬達
		Roller_Fwd := TRUE;
		bDone := TRUE;
		step := 0;
		
	
		


	720:
		Roller_Fwd := FALSE;
		IF IO.i112 THEN
			// 滾輪馬達保護氣跳脫
			step := step + 10000;
		ELSE
			step := step + 1;
		END_IF
		
	721:
		Roller_Rev := TRUE;
		bDone := TRUE;
		step := 0;
		
	
		


	780:
		Roller_Rev := FALSE;
		Roller_Fwd := FALSE;
		bDone := TRUE;
		step := 0;
END_CASE
END_ACTION

ACTION step_8_Jog_UpDown:
CASE step OF
	800:
		Roller_Up 	:= TRUE;
		Roller_Down := FALSE;
		
		tmr1.PT := T#10S;
		tmr1.IN := TRUE;
		step := step + 1;
		
	801: // 滾輪上升
		IF NOT IO.i315 OR tmr1.Q THEN
			Roller_Up := FALSE;
			tmr1.IN := FALSE;
			IF not IO.i315 THEN
				step := step + 1;
			ELSE
				// 上升超時
				step := step + 10000;
			END_IF
		END_IF
		
	802:
		bDone := TRUE;
		step := 0;
		
	
		


	820:
		Roller_Up := FALSE;
		Roller_Down := TRUE;
		
		tmr1.PT := T#10S;
		tmr1.IN := TRUE;
		step := step + 1;
		
	821: // 滾輪上升
		IF IO.i315 OR tmr1.Q THEN
			Roller_Down := FALSE;
			tmr1.IN := FALSE;
			IF IO.i315 THEN
				step := step + 1;
			ELSE
				// 上升超時
				step := step + 10000;
			END_IF
		END_IF
		
	822:
		bDone := TRUE;
		step := 0;
		
	

END_CASE
END_ACTION

END_PROGRAM

// ---- POUs/資料轉換/HMI_WEB_dataConver.TcPOU
PROGRAM HMI_WEB_dataConver
VAR
END_VAR

Hmi_Web.Car_pos := Axis.FeedCar.Pos;

END_PROGRAM

// ---- POUs/硬體控制/台車/編碼器/MM540.TcPOU
FUNCTION_BLOCK MM540
VAR_INPUT
END_VAR
VAR_OUTPUT
	// 等待觸發中
	bActive : BOOL;
	// 忙碌中
	bBuzy : BOOL;
	// 已完成
	bDone : BOOL;
	// 發生錯誤
	bError : BOOL;
END_VAR
VAR
	FeedCar_Enc_raw : MM540_Raw;
	
	Step : INT;
	
	_SetPos : DINT;
	
	_timeout	: TIME := T#10S;
	
	_timeTmr	: TON;
END_VAR

bBuzy := Step > 0 AND Step < 10000;
bActive := FeedCar_Enc_raw.Inc_Preload_Trigger > 0 AND bBuzy;
bError := Step >= 10000;

CASE Step OF
	1000: // 相關暫存器復位
		FeedCar_Enc_raw.Inc_Preload_Trigger := 0;
		bDone := FALSE;
		bActive := TRUE;
		step := step + 1;
		
	1001:
		IF NOT FeedCar_Enc_raw.Inc_Preload_Done THEN
			step := step + 1;
		END_IF
		
	1002:
		step := 1010;
		
		
	1010: // 放置要設定的值
		FeedCar_Enc_raw.Inc_Preload_Value := _SetPos;
		step := step + 1;
		
	1011:
		FeedCar_Enc_raw.Inc_Preload_Trigger := 2;
		_timeTmr.IN := TRUE;
		step := step + 1;
		
	1012:
		IF FeedCar_Enc_raw.Inc_Preload_Done OR _timeTmr.Q THEN 
			
			FeedCar_Enc_raw.Inc_Preload_Trigger := 0;
			_timeTmr.IN := FALSE;
			bActive := FALSE;
			
			// 歸零完成
			IF FeedCar_Enc_raw.Inc_Preload_Done THEN
				step := 1020;
			// 歸零超時
			ELSIF _timeTmr.Q THEN
				step := 1050;
			END_IF
		END_IF
		
	1020:// 歸零完成
		bdone := TRUE;
		step := 0;
		
		
	1050: // 歸零超時
		step := 10000;
END_CASE



_timeTmr(PT:=_timeout);

PROPERTY Buzy : bool
GET
Buzy := bbuzy;
END_GET
END_PROPERTY

PROPERTY Done : bool
GET
Done := bdone;
END_GET
END_PROPERTY

PROPERTY Error : bool
GET
Error := bError;
END_GET
END_PROPERTY

PROPERTY Pos : REAL
GET
Pos := DINT_TO_REAL(FeedCar_Enc_raw.Inc);
END_GET
END_PROPERTY

METHOD SetPos : BOOL
VAR_INPUT
	Pos : DINT;
END_VAR
_SetPos := Pos;

step := 1000;
END_METHOD

END_FUNCTION_BLOCK

// ---- POUs/硬體控制/台車/Axis_VFD.TcPOU
FUNCTION_BLOCK Axis_VFD IMPLEMENTS I_Axis
VAR_INPUT
END_VAR
VAR_OUTPUT
END_VAR
VAR
	// 模式
	Mode: ActionMode;
	// 步進
	step: INT;
	// 發生錯誤步
	ws_step: WSTRING;
	// 目標位置
	TargetPos: LREAL;
	// 動作速度
	Velocity: LREAL;
	
	
(*=======================================
				計時器
=======================================*)
	
	tmr1: TON := (PT := TIME#100MS);
	tmr2: TON := (PT := TIME#100MS);
	tmr100: TON;
	tmr200: TON := (PT := TIME#1S);
	tmr201: TON := (PT := TIME#1S);
	tmr800: TON := (PT := TIME#100MS);
	
	// 超時監視計時器
	tmrWdt: Ton := (PT := TIME#10S0MS);
  	
	
(*=======================================
				軸IO
=======================================*)
	// 原點
	_Origin				: POINTER TO  BOOL;
	
	// 正極限
	_P_Limit			: POINTER TO  BOOL;
	// 負極限
	_N_Limit			: POINTER TO  BOOL;

	// 編碼器
	_Enc : POINTER TO  MM540;
	
	// 變頻器IO
	Axis1_IO: VFD_E_IO;
	
	Limit_status : WORD;
	
	Estop_Old: BOOL;
	
	Estop_Trig : R_TRIG;

(*==============================================*)

	Origin_pos: LREAL;
	// 位置
	_pos : LREAL;
	
	// 軸名稱
	scAxisName : WSTRING;
	
	
	// 位置誤差量
	_ErrorPos: LREAL;
	
	HightSpeed_Error : LREAL := 470;
	MidSpeed_Error : LREAL := 80;
	
	// 上次位置
	_lastPos: LREAL;
	// 速度
	_speed: LREAL;
	
	// 速度
	_speed_average: ARRAY [0..10] OF LREAL;
	
	i : INT;
END_VAR

VAR_OUTPUT
	// 功能執行中
	bBuzy 	: BOOL;
	// 功能結束
	bDone	: BOOL;
	// 發生錯誤
	bError	: BOOL;
	// 錯誤步驟
	iErrorID	: INT;
	// 功能錯誤碼
	iFbErrorID	: INT;
	// 已歸零
	bHome	: BOOL;
	
	rFindPos : LREAL;
END_VAR

VAR_INPUT
	bJogMode: BOOL;
	
	// 負極限
	inLimiter: BOOL;
	// 正極限
	outLimiter: BOOL;
	// 原點
	origin : BOOL;
	
END_VAR

Main();

METHOD AbsMove : BOOL
VAR_INPUT
	// 目標位置
	_Position : LREAL;
	// 移動速度
	_Velocity : LREAL := 0;
END_VAR
bDone := FALSE;
step:=1;
Mode := ActionMode.AbsMove;
TargetPos := _Position;
Velocity := _Velocity;
END_METHOD

PROPERTY Buzy : bool
GET
Buzy := bBuzy;
END_GET
END_PROPERTY

PROPERTY Done : bool
GET
Done := bDone;
END_GET
END_PROPERTY

PROPERTY Encoder : LWORD;
SET
_enc := Encoder;
END_SET
END_PROPERTY

PROPERTY Error : bool
GET
Error := bError;
END_GET
END_PROPERTY

METHOD Find : BOOL
VAR_INPUT
END_VAR
bDone := FALSE;
step:=1;
Mode := ActionMode.Find;
END_METHOD

METHOD Homing : BOOL
VAR
END_VAR
bDone := FALSE;
step:=1;
Mode := ActionMode.Home;
END_METHOD

ACTION Main:
Estop_Trig(CLK:= SystemError OR Input.Feed_Reset);

IF Estop_Trig.Q THEN
	iErrorId := step;
	step:=800;
	bDone := FALSE;
END_IF

bBuzy := step > 0 AND step < 10000;
berror := step >= 10000;
IF bBuzy OR berror THEN
	bDone := FALSE;
END_IF

IF bError THEN
	iErrorID := step - 10000;
	Axis1_IO.o_Speed1^ 		:= FALSE;
	Axis1_IO.o_Speed2^ 		:= FALSE;
	Axis1_IO.o_Speed3^ 		:= FALSE;
	Axis1_IO.o_FWD^			:= FALSE;
	Axis1_IO.o_REV^			:= FALSE;
END_IF

IF _N_Limit > 0 THEN
	Limit_status.0 := _N_Limit^;
ELSE
	Limit_status.0 := TRUE;
END_IF

IF _P_Limit > 0 THEN
	Limit_status.1 := _P_Limit^;
ELSE
	Limit_status.1 := TRUE;
END_IF

IF _Origin > 0 THEN
	Limit_status.2 := _Origin^;
END_IF



ws_step := INT_TO_WSTRING(step);

CASE step OF
	0://程式待命
		tmr1.IN					:= FALSE;
		tmr100.IN				:= FALSE;
		tmr200.IN				:= FALSE;
		tmr201.IN				:= FALSE;
		tmr800.IN				:= FALSE;
		tmrWdt.in 				:= FALSE;
		Axis1_IO.o_Speed1^ 		:= FALSE;
		Axis1_IO.o_Speed2^ 		:= FALSE;
		Axis1_IO.o_Speed3^ 		:= FALSE;
		Axis1_IO.o_FWD^			:= FALSE;
		Axis1_IO.o_REV^			:= FALSE;
		
END_CASE

_enc^();



_pos := _Enc^.Pos * Config.FeedCar_Enc_Scal;

_speed_average[10] := (_pos - _lastPos) * 100;

FOR i := 0 TO 9 DO
	_speed_average[9 - i] := _speed_average[10 - i];
END_FOR

_speed := 0;

FOR i := 0 TO 10 DO
	_speed := _speed + _speed_average[i];
END_FOR

_speed := _speed / 11;

_lastPos := _pos;

_ErrorPos := TargetPos - _pos;

IF step > 0 THEN
	Step0_Start();
	Step1_1_AbsMove();
//	Step1_2_RelMove();
	Step1_3_Home();
	Step1_4_Find();
	Step8_End();
END_IF




timer();


// 碰到正轉極限
IF NOT Limit_status.0 AND Axis1_IO.o_REV^ THEN
	Axis1_IO.o_REV^ := FALSE;
END_IF

// 碰到反轉極限
IF NOT Limit_status.1 AND Axis1_IO.o_FWD^ THEN
	Axis1_IO.o_FWD^ := FALSE;
END_IF
END_ACTION

PROPERTY Name : WSTRING
GET
Name := scAxisName;
END_GET
SET
scAxisName := Name;
END_SET
END_PROPERTY

PROPERTY Pos : LREAL
GET
Pos := _pos;
END_GET
END_PROPERTY

METHOD PowerOff : BOOL
VAR_INPUT
END_VAR
(*===============================
			關閉馬達
  ===============================*)
step:=800;
END_METHOD

METHOD PowerOn : BOOL
VAR_INPUT
END_VAR
bDone := FALSE;
step:=1;
Mode := ActionMode.DoNothing;
END_METHOD

METHOD RelMove : BOOL
VAR_INPUT
	// 目標位置
	_Position : LREAL;
	
	// 移動速度
	_Velocity : LREAL := 0;
END_VAR
bDone := FALSE;
step:=1;
Mode := ActionMode.RelMove;
TargetPos := _Position;

IF _Velocity = 0 THEN
	Velocity := 10;
ELSE
	Velocity := _Velocity;
END_IF
END_METHOD

METHOD Set_VFD_IO : BOOL
VAR_INPUT
	FWD : LWORD;
	REV : LWORD;
	Speed_Io_1 : LWORD;
	Speed_Io_2 : LWORD;
	Speed_Io_3 : LWORD;
	Reset : LWORD;
	
	Run : LWORD;
	Error : LWORD;
END_VAR
Axis1_IO.o_FWD := FWD;
Axis1_IO.o_REV := REV;
Axis1_IO.o_Speed1 := Speed_Io_1;
Axis1_IO.o_Speed2 := Speed_Io_2;
Axis1_IO.o_Speed3 := Speed_Io_3;
Axis1_IO.o_Reset := Reset;

Axis1_IO.i_Run := RUN;
Axis1_IO.i_Error := Error;
END_METHOD

METHOD SetLimit : BOOL
VAR_INPUT

END_VAR
END_METHOD

METHOD SetLimit_IO : BOOL
VAR_INPUT
	Origin : LWORD;
	
	P_Limit : LWORD;
	
	N_Limit : LWORD;
END_VAR
_Origin := Origin;
_P_Limit := P_Limit;
_N_Limit := N_Limit;
END_METHOD

ACTION Step0_Start:
	(*============================
				啟動馬達
	  ============================*)
CASE step OF
	
	1://開始移動流程
		// 設定狀態
		bDone := FALSE;
		Axis1_IO.o_Reset^ :=FALSE;
		tmrWdt.IN := FALSE;
		IF NOT bDone THEN
			step := 10;
		END_IF
		
	10:
		IF NOT Axis1_IO.i_Error^ THEN
			step := step + 1;
		ELSE
			step := 20;
		END_IF
		
	11:
		Axis1_IO.o_Reset^ :=TRUE;
		step := step + 1;
		
	12:
		tmr1.PT := T#2S;
		tmr1.IN := TRUE;
		IF tmr1.Q OR NOT Axis1_IO.i_Error^ THEN
			tmr1.IN := FALSE;
			step := step + 1;
		END_IF


	13:
		Axis1_IO.o_Reset^ :=FALSE;
		IF NOT Axis1_IO.i_Error^ THEN
			// 變頻器錯誤無法重置		
			step := step + 10000;
		ELSE
			step := 20;
		END_IF
		
	20:
		step := 80;
		
	80: //模式選擇
		CASE Mode OF
			ActionMode.AbsMove:
				step := 100;
				
			ActionMode.RelMove:
				step := 200;
				
			ActionMode.Home:
				step := 300;
				
			ActionMode.Find:
				step		:= 400;
				
			ActionMode.DoNothing:
				step := step + 1;
		END_CASE
		
	81:
		bdone := TRUE;
		step := 0;
		
END_CASE
END_ACTION

ACTION Step1_1_AbsMove:
	(*========================================
					開始移動
	=========================================*)	

	

CASE step OF
	100:		
		Axis1_IO.o_Speed1^ 		:= FALSE;
		Axis1_IO.o_Speed2^ 		:= FALSE;
		Axis1_IO.o_Speed3^ 		:= FALSE;
		step := step + 1;
		
	101:
		IF ABS(_ErrorPos) < 2 THEN 
			step:= 190;
		ELSE
			step := step + 1;
		END_IF
		
	102:
		step:= 109;
		
	109:
		step:= 110;
		

	110: // 設定移動位置
		Axis1_IO.o_Speed3^ := TRUE;
		IF _ErrorPos > 0 THEN
			Axis1_IO.o_FWD^ := TRUE;
			Axis1_IO.o_REV^ := FALSE;
		ELSE
			Axis1_IO.o_FWD^ := FALSE;
			Axis1_IO.o_REV^ := TRUE;
		END_IF
	
	
		IF ABS(_ErrorPos) > config.dis_to_MidSpeed AND (Velocity > 0) THEN
			step := step + 1;
		ELSIF ABS(_ErrorPos) > config.dis_to_LowSpeed THEN
			step := 120;
		ELSE
			step := 130;
		END_IF
		
		
	111:
		Axis1_IO.o_Speed2^ := TRUE;
		step := step + 1;
		
	112:
		IF ABS(_ErrorPos) <= ABS(_speed) * 1.5 THEN
			step:=step + 1;
		END_IF
		
	113:
		step:= 120;
		
	120:
		IF ABS(_ErrorPos) > config.dis_to_LowSpeed THEN
			step:=step + 1;
		ELSE
			step := 130;
		END_IF
		
	121:
		Axis1_IO.o_Speed1^ := TRUE;
		Axis1_IO.o_Speed2^ := FALSE;
		step:=step + 1;
		
	122:
		IF ABS(_ErrorPos) <= config.dis_to_LowSpeed THEN
			step:=step + 1;
		END_IF
		
	123:
		step:= 130;
		
	130:
		Axis1_IO.o_Speed1^ := TRUE;
		Axis1_IO.o_Speed2^ := TRUE;
		
		step:=step + 1;
		
	131:
		IF ABS(_speed) < 20 THEN
			Axis1_IO.o_Speed3^ := FALSE;
		END_IF
		
		IF ABS(_ErrorPos) <= 2 THEN
			Axis1_IO.o_FWD^ := FALSE;
			Axis1_IO.o_REV^ := FALSE;
			Axis1_IO.o_Speed1^ := FALSE;
			Axis1_IO.o_Speed2^ := FALSE;
			step:=step + 1;
		END_IF
		
	132:
		step:= 190;


	190:
		bDone := TRUE;
		step:=0;
END_CASE
END_ACTION

ACTION Step1_2_RelMove:
	(*========================================
					開始移動
	=========================================*)	
CASE step OF
	200:
		fb_RelMove.Execute := FALSE;
		Axis1Halt.Execute := FALSE;
		Axis1Stop.Execute := FALSE;
		step := step + 1;
		
	201:
		IF Velocity = 0 THEN
			pMsg.Push_Error(
				ErrorCodeConver.Str2(scAxisName, ":Rel設定速度為0", 0)
			);
		ELSE
			step := step + 1;
		END_IF
		
	202:
		IF TargetPos = 0 THEN 
			step:= 280;
		ELSE
			step := step + 1;
		END_IF
		
	203:
		IF Axis1.Status.HasJob THEN
			Axis1Halt.Deceleration := 0;
			Axis1Halt.Execute := TRUE;
			step := step + 1;
		ELSE
			step:= 209;
		END_IF
		
	204:
		IF Axis1Halt.Busy OR Axis1Halt.Done OR Axis1Halt.Error THEN
			step:=step + 1;
		END_IF
		
	205:
		IF Axis1Halt.Done THEN
			Axis1Halt.Execute := FALSE;
			step:=step + 1;
		ELSIF Axis1Halt.Error THEN
			Axis1Halt.Execute := FALSE;
			step:=step + 10000;
		END_IF
		
	206:
		step:= 209;
		
	209:
		step:= 210;
		

	210: // 設定移動位置
		fb_RelMove.Distance := TargetPos;
		fb_RelMove.Velocity:= Velocity;
		fb_RelMove.BufferMode:= MC_Aborting;
		step:=step + 1;
		
	211:
		fb_RelMove.Execute := TRUE;
		step:=step + 1;
		
	212:
		IF fb_RelMove.Busy OR fb_RelMove.Done OR fb_RelMove.Error THEN
			step:=step + 1;
		END_IF
		
	213:
		IF fb_RelMove.Done THEN
			fb_RelMove.Execute := FALSE;
			step:=step + 1;
		ELSIF fb_RelMove.Error THEN
			pMsg.Push_Error(
				ErrorCodeConver.Str2(scAxisName, ":Rel移動失敗", fb_RelMove.ErrorID)
			);
			fb_RelMove.Execute := FALSE;
			step:=step + 10000;
		END_IF
		
	214:
		step:=290;
		
	280:
		tmr1.PT := T#500MS;
		tmr1.IN := TRUE;
		IF tmr1.Q THEN
			tmr1.IN := FALSE;
			step:=step + 1;
		END_IF
		
	281:
		step := 290;
		
	290:
		bDone := TRUE;
		step:=890;
END_CASE
END_ACTION

ACTION Step1_3_Home:
(*========================================
				歸零
=========================================*)	
CASE step OF
	// 檢查是否有原點感應器 ， 沒有直接結束歸零
	300:
		
		IF _Origin > 0 THEN
			step := step + 1;
		ELSE
			step := 0;
		END_IF
		
	301:
		Axis1_IO.o_Speed1^	:= FALSE;
		Axis1_IO.o_Speed2^	:= FALSE;
		Axis1_IO.o_Speed3^	:= FALSE;
		Axis1_IO.o_FWD^ 	:= FALSE;
		Axis1_IO.o_REV^ 	:= FALSE;
		step := 310;
		
	310: // 沒原點開關訊號  (開關已碰到)
		IF NOT _Origin^ THEN
			step := step + 1;
		ELSE
			step := 320;
		END_IF
		
	311:
		Axis1_IO.o_Speed1^ := TRUE;
		Axis1_IO.o_FWD^ := TRUE;
		step := step + 1;
		
	312:
		tmr1.PT := T#2S;
		tmr1.IN := TRUE;
		IF tmr1.Q OR _Origin^ THEN
			tmr1.IN := FALSE;
			Axis1_IO.o_FWD^ := FALSE;
			Axis1_IO.o_Speed1^ := FALSE;
	
			IF _Origin^ THEN
				step := step + 1;
			ELSE
		// !!錯誤!!  原點訊號沒出現
				step := step + 10000;
			END_IF
			
		END_IF
		
	313:
		step := 320;
		
	320: // 往反方向找原點開關
		Axis1_IO.o_Speed3^ := TRUE;
		Axis1_IO.o_Speed1^ := TRUE;
		Axis1_IO.o_Rev^ := TRUE;
		step := step + 1;
		
	321:
		tmr1.PT := T#2m;
		tmr1.IN := TRUE;
		IF tmr1.Q OR not _Origin^ THEN
			tmr1.IN := FALSE;
			Axis1_IO.o_Rev^ := FALSE;
			Axis1_IO.o_Speed1^ := FALSE;
	
			IF NOT _Origin^ THEN
				step := step + 1;
			ELSE
		// !!錯誤!!  原點訊號沒消失
				step := step + 10000;
			END_IF
			
		END_IF
		
	322:
		step := 330;
		
	330: // 往 正方向  脫離原點開關 最慢速
		Axis1_IO.o_Speed1^ := TRUE;
		Axis1_IO.o_Speed2^ := TRUE;
		Axis1_IO.o_Speed3^ := FALSE;
		Axis1_IO.o_FWD^ := TRUE;
		step := step + 1;
		
	331:
		tmr1.PT := T#10S;
		tmr1.IN := TRUE;
		IF tmr1.Q OR _Origin^ THEN
			tmr1.IN := FALSE;
			Axis1_IO.o_FWD^ := FALSE;
			Axis1_IO.o_Speed1^ := FALSE;
			Axis1_IO.o_Speed2^ := FALSE;
			IF _Origin^ THEN
				step := step + 1;
			ELSE
		// !!錯誤!!  原點訊號沒恢復
				step := step + 10000;
			END_IF
			
		END_IF
		
	332:
		step := 340;
		
	340:
		tmr1.PT := T#500ms;
		tmr1.IN := TRUE;
		IF tmr1.Q THEN
			tmr1.IN := FALSE;
			step := step + 1;
		END_IF
		
	341:
		_enc^.SetPos(Config.FeedCar_Enc_Origin_offset);
		bhome := FALSE;
		step := step + 1;
		
	342:
		IF _enc^.bActive THEN
			step := step + 1;
		END_IF
		
	343:
		Axis1_IO.o_Speed1^ := TRUE;
		Axis1_IO.o_Speed2^ := TRUE;
		Axis1_IO.o_FWD^ := TRUE;
		step := step + 1;
		
	344:
		IF _enc^.Done OR _enc^.Error THEN
			Axis1_IO.o_Speed1^ := FALSE;
			Axis1_IO.o_Speed2^ := FALSE;
			Axis1_IO.o_FWD^ := FALSE;
			IF _enc^.Done THEN
				step := step + 1;
			ELSIF _enc^.Error THEN
				step := step + 10000;
			END_IF
		END_IF
		
	345:
		bhome := TRUE;
		bdone := TRUE;
		step := 0;
END_CASE
END_ACTION

ACTION Step1_4_Find:
	(*========================================
					開始移動
	=========================================*)	

	

CASE step OF
	400:		
		Axis1_IO.o_Speed1^ 		:= FALSE;
		Axis1_IO.o_Speed2^ 		:= FALSE;
		step := step + 1;
		
	401:
		step := 410;
		
		
	410:
		Axis1_IO.o_Speed1^	:= TRUE;
		Axis1_IO.o_Speed2^	:= FALSE;
		step := step + 1;
		
	411:
		Axis1_IO.o_FWD^ 	:= TRUE;
		step := step + 1;
		
	412:
		tmr1.PT := T#1S;
		tmr1.IN := _speed < 10;
		IF tmr1.Q THEN
			tmr1.IN := FALSE;
			step := step + 1;
		END_IF
		
	413:
		step := 420;
		
		
	420:
		Axis1_IO.o_Speed2^	:= TRUE;
		step := step + 1;
		
	421:
		tmr1.PT := T#0.5S;
		tmr1.IN := _speed < 10;
		IF tmr1.Q THEN
			tmr1.IN := FALSE;
			step := step + 1;
		END_IF
		
	422:
		step := 430;
		
		
	430:
		rFindPos := config.pos_CarPin_StopPoint - _pos;
		step := step + 1;
		
	431:
		Axis1_IO.o_Speed1^	:= TRUE;
		Axis1_IO.o_Speed2^	:= TRUE;
		Axis1_IO.o_FWD^		:= FALSE;
		Axis1_IO.o_REV^		:= TRUE;
		step := step + 1;
		
	432:
		tmr1.PT := T#3S;
		tmr1.IN := TRUE;
		IF tmr1.Q THEN
			tmr1.IN := FALSE;
			step := step + 1;
		END_IF
		
	433:
		Axis1_IO.o_Speed1^	:= FALSE;
		Axis1_IO.o_Speed2^	:= FALSE;
		Axis1_IO.o_Speed3^	:= FALSE;
		Axis1_IO.o_FWD^		:= FALSE;
		Axis1_IO.o_REV^		:= FALSE;
		step := step + 1;
		
	434:
		bdone := TRUE;
		step := 0;
END_CASE
END_ACTION

ACTION Step8_End:
	(*======================================
					關閉馬達
	  ======================================*)
CASE step OF
	800:
		Axis1_IO.o_Speed1^	:= FALSE;
		Axis1_IO.o_Speed2^	:= FALSE;
		Axis1_IO.o_Speed3^	:= FALSE;
		Axis1_IO.o_FWD^		:= FALSE;
		Axis1_IO.o_REV^		:= FALSE;
		step := step + 1;
		
	801:
		step := 0;

END_CASE
END_ACTION

METHOD Stop : BOOL
VAR_INPUT
END_VAR
(*===============================
			關閉馬達
  ===============================*)
step:=800;
END_METHOD

ACTION timer:
tmr1();
tmr2();
tmr100(PT:=T#50MS);
tmr200();
tmr201();
tmr800();
tmrWdt();
END_ACTION

END_FUNCTION_BLOCK

// ---- POUs/硬體控制/測高/AxisBase.TcPOU
FUNCTION_BLOCK AxisBase
VAR_INPUT
END_VAR
VAR_OUTPUT
END_VAR
VAR
	// 模式
	Mode: ActionMode;
	// 步進
	step: INT;
	stepA: INT;
	// 發生錯誤步
	ws_step: WSTRING;
	// 目標位置
	TargetPos: LREAL;
	// 動作速度
	Velocity: LREAL;
	// 動作減速度
	Dec : LREAL := 0;
(*=======================================
				計時器
=======================================*)
	
	tmr1: TON := (PT := TIME#100MS);
	tmr2: TON := (PT := TIME#100MS);
	tmr100: TON;
	tmr200: TON := (PT := TIME#1S);
	tmr201: TON := (PT := TIME#1S);
	tmr800: TON := (PT := TIME#100MS);
	
	// 超時監視計時器
	tmrWdt: Ton := (PT := TIME#10S0MS);
  	
	
(*=======================================
				軸IO
=======================================*)

	
	Estop_Old: BOOL;
	
	Estop_Trig : R_TRIG;

(*==============================================
					MC 功能快
==============================================*)
	

	Axis1Power	: MC_Power;
	Axis1Reset	: MC_Reset;
	Axis1Stop	: MC_Stop;
	Axis1Halt	: MC_Halt;
	
	fb_AbsMove	: MC_MoveAbsolute;
	fb_RelMove	: MC_MoveRelative;
	fb_Home		: MC_Home;
	fb_BacklashCompensation	: MC_BacklashCompensation;
	
	fb_Axis1_NcIoOutput : MC_WriteNcIoOutput;
	
	
	fb_WriteBoolParameter : MC_WriteBoolParameterPersistent;
	fb_WriteParameter: MC_WriteParameterPersistent;
(*==============================================*)

	Origin_pos: LREAL;
	
	// 軸名稱
	scAxisName : WSTRING;
END_VAR

VAR_OUTPUT
	// 功能執行中
	bBuzy 	: BOOL;
	// 功能結束
	bDone	: BOOL;
	// 發生錯誤
	bError	: BOOL;
	// 錯誤步驟
	iErrorID	: INT;
	// 功能錯誤碼
	iFbErrorID	: INT;
	// 已歸零
	bHome	: BOOL;
	// 位置
	fPos : LREAL;
END_VAR

VAR_INPUT
	bJogMode: BOOL;
	// 移動軸
	Axis1: REFERENCE TO AXIS_REF;
	// 負極限
	inLimiter: BOOL;
	// 正極限
	outLimiter: BOOL;
	// 原點
	origin : BOOL;
	
	
END_VAR

IF __ISVALIDREF(Axis1) THEN
	Main();
END_IF

METHOD AbsMove : BOOL
VAR_INPUT
	// 目標位置
	_Position : LREAL;
	
	// 移動速度
	_Velocity : LREAL := 0;
END_VAR
bDone := FALSE;
step:=1;
Mode := ActionMode.AbsMove;
TargetPos := _Position;

IF _Velocity = 0 THEN
	Velocity := 10;
ELSE
	Velocity := _Velocity;
END_IF
END_METHOD

PROPERTY Axis_States : ST_AxisStatus
GET
Axis1.ReadStatus();
Axis_States := Axis1.Status;
END_GET
END_PROPERTY

METHOD Homing : BOOL
VAR
END_VAR
bDone := FALSE;
step:=1;
Mode := ActionMode.Home;
END_METHOD

ACTION Main:
Estop_Trig(CLK:= (SystemError OR Estop OR Input.Feed_Reset) AND bBuzy );

IF Estop_Trig.Q THEN
	iErrorId := step;
	step:=800;
	bDone := FALSE;
END_IF

bBuzy := step > 0 AND step < 10000;
berror := step >= 10000;
IF bBuzy OR berror THEN
	bDone := FALSE;
END_IF
IF bError THEN
	iErrorID := step - 10000;
	
END_IF

ws_step := INT_TO_WSTRING(step);

CASE step OF
	0://程式待命
		tmr1.IN					:= FALSE;
		tmr100.IN				:= FALSE;
		tmr200.IN				:= FALSE;
		tmr201.IN				:= FALSE;
		tmr800.IN				:= FALSE;
		tmrWdt.in 				:= FALSE;
		
END_CASE

IF step > 0 THEN
	Step0_Start();
	Step1_1_AbsMove();
	Step1_2_RelMove();
	Step1_3_Home();
	Step8_End();
END_IF

MC_FB();
fPos := LREAL_TO_REAL(Axis1.NcToPlc.ActPos);
timer();
END_ACTION

ACTION MC_FB:
// 正轉極限
Axis1Power.Enable_Positive:= OutLimiter;
// 反轉極限
Axis1Power.Enable_Negative:= inLimiter;

Axis1.ReadStatus();

// 軸速度百分比
Axis1Power.Override := Axis.Override; 


(*===================== 軸電源 =====================*)
Axis1Power(Axis:= Axis1);


(*===================== 軸重置 =====================*)
Axis1Reset(Axis:= Axis1);


(*===================== 軸停止 =====================*)
Axis1Stop(Axis:= Axis1);


(*===================== 軸命令取消 =====================*)
Axis1Halt(Axis:= Axis1);


(*===================== 軸絕對移動 =====================*)
fb_AbsMove(Axis:= Axis1);


(*===================== 軸相對移動 =====================*)
fb_RelMove(Axis:= Axis1);

(*===================== 軸歸零 =====================*)
fb_Axis1_NcIoOutput(Axis:= Axis1, Device := NcIoDeviceDrive, NcIoOutput := NcIoOutputnCtrl2);

(*===================== 軸歸零 =====================*)
fb_Home(Axis:= Axis1, HomingMode:= MC_Direct);

(*===================== 軸寫入BOOL參數 =====================*)
fb_WriteBoolParameter(Axis:= Axis1);

(*===================== 軸寫入參數 =====================*)
fb_WriteParameter(Axis:= Axis1);

(*===================== 背隙補償 =====================*)
fb_BacklashCompensation(Axis:= Axis1);
END_ACTION

PROPERTY Name : WSTRING
GET
Name := scAxisName;
END_GET
SET
scAxisName := Name;
END_SET
END_PROPERTY

PROPERTY Pos : LREAL
GET
pos := fPos;
END_GET
END_PROPERTY

METHOD PowerOff : BOOL
VAR_INPUT
END_VAR
(*===============================
			關閉馬達
  ===============================*)
step:=800;
END_METHOD

METHOD PowerOn : BOOL
VAR_INPUT
END_VAR
bDone := FALSE;
step:=1;
Mode := ActionMode.DoNothing;
END_METHOD

METHOD RelMove : BOOL
VAR_INPUT
	// 目標位置
	_Position : LREAL;
	
	// 移動速度
	_Velocity : LREAL := 0;
END_VAR
bDone := FALSE;
step:=1;
Mode := ActionMode.RelMove;
TargetPos := _Position;

IF _Velocity = 0 THEN
	Velocity := 10;
ELSE
	Velocity := _Velocity;
END_IF
END_METHOD

METHOD SetDyn : BOOL
VAR_INPUT
	SetJog : BOOL;
END_VAR
//IF SetJog THEN
//	fb_AbsMove.Acceleration := SpdC.DnZ_Jog_Accelerated;
//	fb_AbsMove.Deceleration := SpdC.DnZ_Jog_Deceleration;
//	fb_RelMove.Acceleration := SpdC.DnZ_Jog_Accelerated;
//	fb_RelMove.Deceleration := SpdC.DnZ_Jog_Deceleration;
//ELSE
//	fb_AbsMove.Acceleration := SpdC.DnZ_Accelerated;
//	fb_AbsMove.Deceleration := SpdC.DnZ_Deceleration;
//	fb_RelMove.Acceleration := SpdC.DnZ_Accelerated;
//	fb_RelMove.Deceleration := SpdC.DnZ_Deceleration;
//end_if
END_METHOD

METHOD SetLimit : BOOL
VAR_INPUT
END_VAR
stepA := 1;
END_METHOD

ACTION Step0_Start:
	(*============================
				啟動馬達
	  ============================*)
CASE step OF
	
	1://開始移動流程
		// 設定狀態
		bDone := FALSE;
		tmrWdt.IN := FALSE;
//		SetDyn(bJogMode);
		Axis1Reset.Execute :=FALSE;
		
		IF NOT bDone THEN
			step := 10;
		END_IF
		
	10:
		IF axis1.Status.Error THEN
			step := step + 1;
		ELSE
			step := 20;
		END_IF
		
	11:
		Axis1Reset.Execute :=TRUE;
		step := step + 1;
		
	12:
		IF NOT axis1.Status.Error AND Axis1Reset.Done THEN
			Axis1Reset.Execute :=FALSE;
			step := 20;
		ELSIF Axis1Reset.Error THEN
			pMsg.Push_Error(
				ErrorCodeConver.Str2(scAxisName, ": 馬達無法重置", Axis1Reset.ErrorID)
			);
			Axis1Reset.Execute :=FALSE;
			step:=step + 10000;
		END_IF
		
	20: // 檢查馬達1是否已啟動
		IF NOT Axis1Power.Status  THEN
			step := step + 1;
		ELSE
			step := 60;
		END_IF
		
	21:// 啟動馬達1
		Axis1Power.Enable := TRUE;
		tmrWdt.IN := TRUE;
		step := step + 1;
		
	22:// 等待馬達啟動完成
		IF Axis1Power.Status THEN
			step := step + 1;
			tmrWdt.IN := FALSE;
			
		ELSIF tmrWdt.Q OR Axis1Power.Error THEN
			pMsg.Push_Error(
				ErrorCodeConver.Str2(scAxisName, ":啟動失敗", Axis1Power.ErrorID)
			);
			tmrWdt.IN := FALSE;
			step:=step + 10000;
		END_IF
		
	23:// 馬達啟動後延遲
		tmr1.in:=TRUE;
		IF tmr1.Q THEN
			tmr1.IN:=FALSE;
			step:=60;
		END_IF
		
	
			

	60: 
		fb_BacklashCompensation.Enable := FALSE;
		step := step + 1;
		
		
	61:	
		// 背隙值 (mm)
		fb_BacklashCompensation.Backlash := 0.05;
		// 正向補償 (往正方向移動時補償，預設是反方向移動時補償)
		fb_BacklashCompensation.CompensationInPositiveDirection := FALSE;
		// 背隙補償的速度 (mm/s)
		fb_BacklashCompensation.Ramp := 1;
		// 解除時機
		fb_BacklashCompensation.DisableMode  := E_DisableMode.DisableModeReset;
		// 功能啟動
		fb_BacklashCompensation.Enable := TRUE;
		step := step + 1;
		
	62:
		IF fb_BacklashCompensation.Enabled THEN
			step := step + 1;
		ELSIF fb_BacklashCompensation.Error THEN
			fb_BacklashCompensation.Enable := FALSE;
			step := step + 1;
		END_IF
		
	63:
		step := 80;
		
	80: //模式選擇
		CASE Mode OF
			ActionMode.AbsMove:
				step := 100;
				
			ActionMode.RelMove:
				step := 200;
				
			ActionMode.Home:
				step := 300;
				
			ActionMode.Find:
				step := 400;
				
			ActionMode.DoNothing:
				step := step + 1;
		END_CASE
		
	81:
		bdone := TRUE;
		step := 0;
		
END_CASE
END_ACTION

ACTION Step1_1_AbsMove:
	(*========================================
					開始移動
	=========================================*)	
CASE step OF
	100:
		fb_AbsMove.Execute := FALSE;
		Axis1Halt.Execute := FALSE;
		Axis1Stop.Execute := FALSE;
		step := step + 1;
		
	101:
		IF Velocity = 0 THEN
			pMsg.Push_Error(
				ErrorCodeConver.Str2(scAxisName, ":Abs設定速度為0", 0)
			);
		ELSE
			step := step + 1;
		END_IF
		
	102:
		IF fPos > TargetPos - 0.1 AND fPos < TargetPos + 0.1 THEN 
			step:= 190;
		ELSE
			step := step + 1;
		END_IF
		
	103:
		IF Axis1.Status.HasJob THEN
			Axis1Halt.Deceleration := 0;
			Axis1Halt.Execute := TRUE;
			step := step + 1;
		ELSE
			step:= 109;
		END_IF
		
	104:
		IF Axis1Halt.Busy OR Axis1Halt.Done OR Axis1Halt.Error THEN
			step:=step + 1;
		END_IF
		
	105:
		IF Axis1Halt.Done THEN
			Axis1Halt.Execute := FALSE;
			step:=step + 1;
		ELSIF Axis1Halt.Error THEN
			Axis1Halt.Execute := FALSE;
			step:=step + 10000;
		END_IF
		
	106:
		step:= 109;
		
	109:
		step:= 110;
		

	110: // 設定移動位置
		fb_AbsMove.Position := TargetPos;
		fb_AbsMove.Velocity:= Velocity;
		fb_AbsMove.BufferMode:= MC_Aborting;
		step:=step + 1;
		
	111:
		fb_AbsMove.Execute := TRUE;
		step:=step + 1;
		
	112:
		IF fb_AbsMove.Busy OR fb_AbsMove.Done OR fb_AbsMove.Error THEN
			step:=step + 1;
		END_IF
		
	113:
		IF fb_AbsMove.Done OR (TargetPos <= 0 AND pos < 2 AND Origin) THEN
			fb_AbsMove.Execute := FALSE;
			step:=step + 1;
		ELSIF fb_AbsMove.Error THEN
			pMsg.Push_Error(
				ErrorCodeConver.Str2(scAxisName, ":Abs移動失敗", fb_AbsMove.ErrorID)
			);
			fb_AbsMove.Execute := FALSE;
			step:=step + 10000;
		END_IF
		
	114:
		step := 190;
		
	190:
		bDone := TRUE;
		step:=890;
END_CASE
END_ACTION

ACTION Step1_2_RelMove:
	(*========================================
					開始移動
	=========================================*)	
CASE step OF
	200:
		fb_RelMove.Execute := FALSE;
		Axis1Halt.Execute := FALSE;
		Axis1Stop.Execute := FALSE;
		step := step + 1;
		
	201:
		IF Velocity = 0 THEN
			pMsg.Push_Error(
				ErrorCodeConver.Str2(scAxisName, ":Rel設定速度為0", 0)
			);
		ELSE
			step := step + 1;
		END_IF
		
	202:
		IF TargetPos = 0 THEN 
			step:= 280;
		ELSE
			step := step + 1;
		END_IF
		
	203:
		IF Axis1.Status.HasJob THEN
			Axis1Halt.Deceleration := 0;
			Axis1Halt.Execute := TRUE;
			step := step + 1;
		ELSE
			step:= 209;
		END_IF
		
	204:
		IF Axis1Halt.Busy OR Axis1Halt.Done OR Axis1Halt.Error THEN
			step:=step + 1;
		END_IF
		
	205:
		IF Axis1Halt.Done THEN
			Axis1Halt.Execute := FALSE;
			step:=step + 1;
		ELSIF Axis1Halt.Error THEN
			Axis1Halt.Execute := FALSE;
			step:=step + 10000;
		END_IF
		
	206:
		step:= 209;
		
	209:
		step:= 210;
		

	210: // 設定移動位置
		fb_RelMove.Distance := TargetPos;
		fb_RelMove.Velocity:= Velocity;
		fb_RelMove.BufferMode:= MC_Aborting;
		step:=step + 1;
		
	211:
		fb_RelMove.Execute := TRUE;
		step:=step + 1;
		
	212:
		IF fb_RelMove.Busy OR fb_RelMove.Done OR fb_RelMove.Error THEN
			step:=step + 1;
		END_IF
		
	213:
		IF fb_RelMove.Done THEN
			fb_RelMove.Execute := FALSE;
			step:=step + 1;
		ELSIF fb_RelMove.Error THEN
			pMsg.Push_Error(
				ErrorCodeConver.Str2(scAxisName, ":Rel移動失敗", fb_RelMove.ErrorID)
			);
			fb_RelMove.Execute := FALSE;
			step:=step + 10000;
		END_IF
		
	214:
		step:=290;
		
	280:
		tmr1.PT := T#500MS;
		tmr1.IN := TRUE;
		IF tmr1.Q THEN
			tmr1.IN := FALSE;
			step:=step + 1;
		END_IF
		
	281:
		step := 290;
		
	290:
		bDone := TRUE;
		step:=890;
END_CASE
END_ACTION

ACTION Step1_3_Home:
(*========================================
				歸零
=========================================*)	
CASE step OF
	300:
		fb_Home.Execute := FALSE;
		step := step + 1;
		
	301:
		Origin_pos := Pos;
		step:= 310;
		
	310: // 尋找負極限訊號
		fb_RelMove.Distance := -9999;
		fb_RelMove.Velocity:= 40;
		fb_RelMove.BufferMode:= MC_Aborting;
		fb_RelMove.Execute := TRUE;
		step:=step + 1;
		
	311:
		IF origin OR fb_RelMove.Busy OR fb_RelMove.Error THEN
			fb_RelMove.Execute := FALSE;
			step:=step + 1;
		END_IF
		
	312:
		IF origin THEN
			Axis1Halt.Execute := TRUE;
			step:=step + 1;
		ELSIF fb_RelMove.Done THEN
			pmsg.Push_Error(ErrorCodeConver.Str2(scAxisName, ":無法找到負極限訊號", 0));
			step:=step + 10000;
		ELSIF fb_RelMove.Error THEN
			pmsg.Push_Error(ErrorCodeConver.Str2(scAxisName, ":歸零移動時發生錯誤", fb_RelMove.ErrorID));
			step:=step + 10000;
		END_IF
		
	313:
		IF Axis1Halt.Busy OR Axis1Halt.Error THEN
			Axis1Halt.Execute := FALSE;
			step:=step + 1;
		END_IF
		
	314:
		IF Axis1Halt.Done THEN
			step:=step + 1;
		ELSIF Axis1Halt.Error THEN
			pmsg.Push_Error(ErrorCodeConver.Str2(scAxisName, ":取消軸移動命令時發生錯誤", Axis1Halt.ErrorID));
			step:=step + 10000;
		END_IF
		
	315:
		tmr200.in :=TRUE;
		IF tmr200.q THEN
			tmr200.in :=FALSE;
			step := step + 1;
		END_IF
		
	316:
		step := 320;
		
		
	320: // 脫離負極限
		fb_RelMove.Distance := 9999;
		fb_RelMove.Velocity:= 5;
		fb_RelMove.BufferMode:= MC_Aborting;
		fb_RelMove.Execute := TRUE;
		step:=step + 1;
		
	321:
		IF fb_RelMove.Busy OR fb_RelMove.Error THEN
			fb_RelMove.Execute := FALSE;
			step:=step + 1;
		END_IF
		
	322:
		IF NOT origin THEN
			Axis1Halt.Execute := TRUE;
			step:=step + 1;
		ELSIF fb_RelMove.Done THEN
			pmsg.Push_Error(ErrorCodeConver.Str2(scAxisName, ":無法找到負極限訊號", 0));
			step:=step + 10000;
		ELSIF fb_RelMove.Error THEN
			pmsg.Push_Error(ErrorCodeConver.Str2(scAxisName, ":歸零移動時發生錯誤", fb_RelMove.ErrorID));
			step:=step + 10000;
		END_IF
		
	323:
		IF Axis1Halt.Busy OR Axis1Halt.Error THEN
			Axis1Halt.Execute := FALSE;
			step:=step + 1;
		END_IF
		
	324:
		IF Axis1Halt.Done THEN
			step:=step + 1;
		ELSIF Axis1Halt.Error THEN
			pmsg.Push_Error(ErrorCodeConver.Str2(scAxisName, ":取消軸移動命令時發生錯誤", Axis1Halt.ErrorID));
			step:=step + 10000;
		END_IF
		
	325:
		tmr200.in :=TRUE;
		IF tmr200.q THEN
			tmr200.in :=FALSE;
			step := step + 1;
		END_IF
		
	326:
		step := 330;
		
	330:
		fb_RelMove.Distance := -9999;
		fb_RelMove.Velocity:= 0.25;
		fb_RelMove.BufferMode:= MC_Aborting;
		fb_RelMove.Execute := TRUE;
		step:=step + 1;
		
	331:
		IF fb_RelMove.Busy OR fb_RelMove.Error THEN
			step:=step + 1;
		END_IF
		
	332:
		IF origin THEN
			Axis1Halt.Execute := TRUE;
			step:=step + 1;
		ELSIF fb_RelMove.Done THEN
			pmsg.Push_Error(ErrorCodeConver.Str2(scAxisName, ":無法找到負極限訊號", 0));
			step:=step + 10000;
		ELSIF fb_RelMove.Error THEN
			pmsg.Push_Error(ErrorCodeConver.Str2(scAxisName, ":歸零移動時發生錯誤", fb_RelMove.ErrorID));
			step:=step + 10000;
		END_IF
		
	333:
		tmr200.in :=TRUE;
		IF tmr200.q THEN
			tmr200.in :=FALSE;
			step := step + 1;
		END_IF
		
	334:
		step := 350;
		
// 	340:
// 		fb_Axis1_NcIoOutput.BitSelectMask := 128;
// 		fb_Axis1_NcIoOutput.BitValues := 128;
// 		fb_Axis1_NcIoOutput.Execute := TRUE;
// 		IF fb_Axis1_NcIoOutput.Done THEN
// 			step := step + 1;
// 			fb_Axis1_NcIoOutput.Execute := FALSE;
// 		ELSIF fb_Axis1_NcIoOutput.Error THEN
// 			pMsg.Push_Error(
// 				ErrorCodeConver.Str3(scAxisName, ":Home寫入驅動器失敗", ws_step, Axis1Halt.ErrorID)
// 			);
// 			fb_Axis1_NcIoOutput.Execute := FALSE;
// 			step:=step + 10000;
// 		END_IF
// 		
// 	341:
// 		fb_Axis1_NcIoOutput.BitSelectMask := 128;
// 		fb_Axis1_NcIoOutput.BitValues := 0;
// 		fb_Axis1_NcIoOutput.Execute := TRUE;
// 		IF fb_Axis1_NcIoOutput.Done THEN
// 			step := step + 1;
// 			fb_Axis1_NcIoOutput.Execute := FALSE;
// 		ELSIF fb_Axis1_NcIoOutput.Error THEN
// 			pMsg.Push_Error(
// 				ErrorCodeConver.Str3(scAxisName, ":Home寫入驅動器失敗", ws_step, Axis1Halt.ErrorID)
// 			);
// 			fb_Axis1_NcIoOutput.Execute := FALSE;
// 			step:=step + 10000;
// 		END_IF
// 		
// 	342:
// 		tmr200.in :=TRUE;
// 		IF tmr200.q THEN
// 			tmr200.in :=FALSE;
// 			step := step + 1;
// 		END_IF
// 		
// 	343:
// 		Axis1Power.Enable := FALSE;
// 		tmrWdt.IN := TRUE;
// 		IF NOT Axis1Power.Status THEN
// 			step := step + 1;
// 			tmrWdt.IN := FALSE;
// 			
// 		ELSIF tmrWdt.Q OR Axis1Power.Error THEN
// 			pMsg.Push_Error(
// 				ErrorCodeConver.Str3(scAxisName, ":關閉失敗", ws_step, Axis1Power.ErrorID)
// 			);
// 			step:=step + 10000;
// 		END_IF	
// 		
// 	344:
// 		tmr200.in :=TRUE;
// 		IF tmr200.q THEN
// 			tmr200.in :=FALSE;
// 			step := step + 1;
// 		END_IF
// 		
// 	345:
// 		step:= 350;
		
	
			
		
	350:// 設定原點
		fb_Home.Execute := TRUE;
		step:=step + 1;
		
	351:
		IF fb_Home.Done THEN
			fb_Home.Execute := FALSE;
			bHome := TRUE;
			step:=step + 1;
		ELSIF fb_Home.Error THEN
			pMsg.Push_Error(
				ErrorCodeConver.Str3(scAxisName, ":位置清除失敗", ws_step, fb_Home.ErrorID)
			);
			fb_Home.Execute := FALSE;
			step:=step + 10000;
		END_IF
		
	352:
		Axis1Power.Enable := TRUE;
		tmrWdt.IN := TRUE;
		IF Axis1Power.Status THEN
			step := step + 1;
			tmrWdt.IN := FALSE;
		ELSIF tmrWdt.Q OR Axis1Power.Error THEN
			pMsg.Push_Error(
				ErrorCodeConver.Str3(scAxisName, ":啟動失敗", ws_step, Axis1Power.ErrorID)
			);
			step:=step + 10000;
		END_IF	
			
	353:
		tmr200.in :=TRUE;
		IF tmr200.q THEN
			tmr200.in :=FALSE;
			step:=step + 1;
		END_IF
		
	354:
		step:= 360;
		
	360:// 設定移動位置
		step:= 390;
	
			
	390://延遲
		tmr200.in :=TRUE;
		IF tmr200.q THEN
			tmr200.in :=FALSE;
			bDone := TRUE;
			step:=890;
		END_IF
END_CASE
END_ACTION

ACTION Step8_End:
	(*======================================
					關閉馬達
	  ======================================*)
CASE step OF
	800:
		Axis1Reset.Execute	:= FALSE;
		Axis1Stop.Execute	:= FALSE;
		Axis1Halt.Execute	:= FALSE;
		fb_AbsMove.Execute	:=FALSE;
		fb_RelMove.Execute	:=FALSE;
		fb_Home.Execute		:=FALSE;
		step := step + 1;
			
	// ============== 停止 + 關閉==============
	801:
		IF Axis1.Status.Moving THEN
			step := step + 1;
		ELSE
			step := 810;
		END_IF
	
	802:
		Axis1Stop.Execute := TRUE;
		step := step + 1;
		
	803:
		Axis1Stop.Execute := TRUE;
		step := step + 1;
		
	804:
		IF Axis1Stop.Done OR Axis1Stop.Error THEN
			Axis1Stop.Execute := FALSE;
			step := step + 1;
		END_IF
		
	805:
		tmr800.PT := T#1S;
		tmr800.in:=TRUE;
		IF tmr800.Q THEN
			tmr800.IN:=FALSE;
			step := step + 1;
		END_IF
		
	806:
		step:=810;
		
	810:
		Axis1Power.Enable := FALSE;
		IF Axis1.Status.Disabled THEN
			step := step + 1;
		END_IF
		
			
	811:// 馬達關閉後延遲
		tmr800.in:=TRUE;
		IF tmr800.Q THEN
			tmr800.IN:=FALSE;
			step := step + 1;
		END_IF
		
	812:
		Mode := ActionMode.DoNothing;
		step:=890;
		
		
// ==============停止==============
	850:
		Axis1Stop.Deceleration := Dec;
		Axis1Stop.Execute := FALSE;
		step := step + 1;
		
	851:
		Axis1Stop.Execute := TRUE;
		step := step + 1;
		
	852:
		IF Axis1Stop.Done OR Axis1Stop.Error THEN
			Axis1Stop.Execute := FALSE;
			step := step + 1;
		END_IF
		
	853:
		tmr800.PT := T#1S;
		tmr800.in:=TRUE;
		IF tmr800.Q THEN
			tmr800.IN:=FALSE;
			step := step + 1;
		END_IF
		
	854:
		step:=890;
		
		
			
	890:// 結束程式
		Mode := ActionMode.DoNothing;
		step:=0;

END_CASE
END_ACTION

METHOD Stop : BOOL
VAR_INPUT
	Dec : LREAL := 0;
END_VAR
(*===============================
			關閉馬達
  ===============================*)
step:=850;
END_METHOD

ACTION timer:
tmr1();
tmr2();
tmr100(PT:=T#50MS);
tmr200();
tmr201();
tmr800();
tmrWdt();
END_ACTION

END_FUNCTION_BLOCK

// ---- MSG/通知訊息/uuidv7_g.TcPOU
PROGRAM uuidv7_g
VAR
	fbStartProcess : NT_StartProcess;
	step: INT;
END_VAR
VAR_OUTPUT
	bBuzy : BOOL;
	bDone : BOOL;
	bError : BOOL;
	UUID:STRING(36);
	ErrorID : UDINT;
END_VAR

CASE step OF
	1:
		UUID := '';
		fbStartProcess.START := FALSE;
		step := step + 1;
		
	2:
		fbStartProcess.START := TRUE;
		step := step + 1;
		
	3:
		IF fbStartProcess.BUSY OR fbStartProcess.ERR THEN
			step := step + 1;
		END_IF
		
	4:
		IF NOT fbStartProcess.BUSY AND NOT fbStartProcess.ERR THEN
			fbStartProcess.START := FALSE;
			step := step + 1;
		ELSIF fbStartProcess.ERR THEN
			fbStartProcess.START := FALSE;
			ErrorID := fbStartProcess.ERRID;
			step := step + 10000;
		END_IF
		
	5:
		IF Len(UUID) >= 36 THEN
			bDone := TRUE;
			step := 0;
		END_IF
END_CASE
	

bBuzy := step > 0 AND step < 10000;

bError := step > 10000;

IF bBuzy THEN
	bDone := FALSE;
END_IF

fbStartProcess(
		NETID := '',
		PATHSTR := 'C:\custom\uuidv7generator_ads\uuidv7generator_ads.exe',
		DIRNAME := 'C:\custom\uuidv7generator_ads',
		COMNDLINE := '127.0.0.1.1.1 851 uuidv7_g.UUID',
		TMOUT := T#1S
	);

METHOD Get
VAR_INPUT
END_VAR
step := 1;
END_METHOD

END_PROGRAM

// ---- Note.TcPOU
PROGRAM Note
VAR
END_VAR

進料台車:
	編碼器對應實際距離: 0.025mm/p
	歸零偏移 : 22mm  > 880p
	最大行程 編碼器 108466 p 實際 2710 mm
	進料範圍 0 - 1000
	暫存範圍 1300 - 2800
	
	30HZ = 164mm/S
	 3HZ =  16mm/S
	 
進料流程:
1.將進料區的工件全部往定位住靠邊，這時候順便檢查 總和寬度 與設定的 容許誤差 做比較
2.將進料區的工件搬移到 等待區 ， 並做分料的動作。
3.將第1支搬入進料區
4.1. 台車繼續 將後續的工件 向前搬 
4.2.1 進料區做工件靠邊
4.2.2 檢測翼板高度，並向前送入雷射機
4.2.3 檢測工件寬度

5.完成進料動作


備註:
緩衝區進完最後的工件後，將再次從1開始


進料計算筆記
	臺車總長 = 1100
	
	工件待命位置= 1400
	
	第二支料分離起始位置 =  工件待命位置 + 臺車寬度 - (第一支料寬 + (第二支料寬 / 2))
	
	第二支料分離結束位置 =  工件待命位置 + 臺車寬度 - (第一支料寬 + 第二支料寬 + 材料排列間距)
	
	第三支料分離起始位置 =  工件待命位置 + 臺車寬度 - (第一支料寬 + 第二支料寬 + (第三支料寬 / 2))
	
	第三支料分離結束位置 =  工件待命位置 + 臺車寬度 - (第二支料分離結束位置 + 第三支料寬 + 材料排列間距)
	
	動作: 從最後一隻開始移動，依序往前


給料計算 筆記
	臺車總長 = 1100
	
	工件待命位置= 1400

	第一支進料移動起始位置 =  工件待命位置 + 臺車寬度 - (第一支料寬 + 材料排列間距)
	
	移動距離 = 給料位置 - 第一支進料移動起始位置
	
	移動次數 = (臺車總長 / 移動距離) ->> 取整數 ，若無小數點，直接減一

END_PROGRAM

// ---- POUs/功能塊/EtherCat相關/EtherCat_Driver_Reset.TcPOU
PROGRAM EtherCat_Driver_Reset
VAR
	step: INT;
END_VAR

VAR_OUTPUT
	bBuzy: BOOL;
	bError: BOOL;
	bDone: BOOL;
	iErrorId : INT;
END_VAR

bBuzy := step > 0 AND step < 10000;
bError := step >= 10000;

// 緊急狀態
IF (EStop OR SystemError) THEN
	bDone := FALSE;
	IF bBuzy THEN
		step := step  + 10000;
	END_IF
END_IF

IF ProgramReset THEN
	iErrorId := step;
	step := 0;
END_IF

CASE step OF
	1:
		bDone := FALSE;
		step := step + 1;
		
	2:
		step := 10;
		
	10:
		IF GetEtherSta.devStates[0].deviceState = 8 THEN
			step := step + 10;
		ELSE
			step := step + 1;
		END_IF
		
	11:
		GetEtherSta.ResetECat1(1001);
		step := step + 1;
		
	12:
		IF GetEtherSta.bBuzy OR GetEtherSta.bError THEN
			step := step + 1;
		END_IF
		
	13:
		IF GetEtherSta.bDone THEN
			step := step + 1;
		ELSIF GetEtherSta.bError THEN
			pMsg.Push_Alarm("重置Driver1-1 EtherCat狀態失敗");
			step := step + 10000;
		END_IF
		
	14:
		step := 20;
		
	20:
		IF GetEtherSta.devStates[1].deviceState = 8 THEN
			step := step + 10;
		ELSE
			step := step + 1;
		END_IF
		
	21:
		GetEtherSta.ResetECat1(1002);
		step := step + 1;
		
	22:
		IF GetEtherSta.bBuzy OR GetEtherSta.bError THEN
			step := step + 1;
		END_IF
		
	23:
		IF GetEtherSta.bDone THEN
			step := step + 1;
		ELSIF GetEtherSta.bError THEN
			pMsg.Push_Alarm("重置Driver1-2 EtherCat狀態失敗");
			step := step + 10000;
		END_IF
		
	24:
		step := 30;
		
	30:
		IF GetEtherSta.devStates[2].deviceState = 8 THEN
			step := step + 10;
		ELSE
			step := step + 1;
		END_IF
		
	31:
		GetEtherSta.ResetECat1(1002);
		step := step + 1;
		
	32:
		IF GetEtherSta.bBuzy OR GetEtherSta.bError THEN
			step := step + 1;
		END_IF
		
	33:
		IF GetEtherSta.bDone THEN
			step := step + 1;
		ELSIF GetEtherSta.bError THEN
			pMsg.Push_Alarm("重置Driver1-3 EtherCat狀態失敗");
			step := step + 10000;
		END_IF
		
	34:
		step := 40;
		
	40:
		IF GetEtherSta.devStates[3].deviceState = 8 THEN
			step := step + 10;
		ELSE
			step := step + 1;
		END_IF
		
	41:
		GetEtherSta.ResetECat1(1004);
		step := step + 1;
		
	42:
		IF GetEtherSta.bBuzy OR GetEtherSta.bError THEN
			step := step + 1;
		END_IF
		
	43:
		IF GetEtherSta.bDone THEN
			step := step + 1;
		ELSIF GetEtherSta.bError THEN
			pMsg.Push_Alarm("重置Driver1-4 EtherCat狀態失敗");
			step := step + 10000;
		END_IF
		
	44:
		step := 50;
		
	50:
		step := 100;
		
// 塔電櫃驅動器
	100:
		IF GetEtherSta.devStates2[5].deviceState = 8 THEN
			step := step + 10;
		ELSE
			step := step + 1;
		END_IF
		
	101:
		GetEtherSta.ResetECat2(1006);
		step := step + 1;
		
	102:
		IF GetEtherSta.bBuzy OR GetEtherSta.bError THEN
			step := step + 1;
		END_IF
		
	103:
		IF GetEtherSta.bDone THEN
			step := step + 1;
		ELSIF GetEtherSta.bError THEN
			pMsg.Push_Alarm("重置Driver2-1 EtherCat狀態失敗");
			step := step + 10000;
		END_IF
		
	104:
		step := 110;
		
	110:
		IF GetEtherSta.devStates2[6].deviceState = 8 THEN
			step := step + 10;
		ELSE
			step := step + 1;
		END_IF
		
	111:
		GetEtherSta.ResetECat2(1007);
		step := step + 1;
		
	112:
		IF GetEtherSta.bBuzy OR GetEtherSta.bError THEN
			step := step + 1;
		END_IF
		
	113:
		IF GetEtherSta.bDone THEN
			step := step + 1;
		ELSIF GetEtherSta.bError THEN
			pMsg.Push_Alarm("重置Driver2-2 EtherCat狀態失敗");
			step := step + 10000;
		END_IF
		
	114:
		step := 120;
	// CarRailln	
	120:
		IF GetEtherSta.devStates2[7].deviceState = 8 THEN
			step := step + 10;
		ELSE
			step := step + 1;
		END_IF
		
	121:
		GetEtherSta.ResetECat2(1008);
		step := step + 1;
		
	122:
		IF GetEtherSta.bBuzy OR GetEtherSta.bError THEN
			step := step + 1;
		END_IF
		
	123:
		IF GetEtherSta.bDone THEN
			step := step + 1;
		ELSIF GetEtherSta.bError THEN
			pMsg.Push_Alarm("重置Driver2-3 EtherCat狀態失敗");
			step := step + 10000;
		END_IF
		
	124:
		step := 130;
		
	130:
		IF GetEtherSta.devStates2[8].deviceState = 8 THEN
			step := step + 10;
		ELSE
			step := step + 1;
		END_IF
		
	131:
		GetEtherSta.ResetECat2(1009);
		step := step + 1;
		
	132:
		IF GetEtherSta.bBuzy OR GetEtherSta.bError THEN
			step := step + 1;
		END_IF
		
	133:
		IF GetEtherSta.bDone THEN
			step := step + 1;
		ELSIF GetEtherSta.bError THEN
			pMsg.Push_Alarm("重置Driver2-4 EtherCat狀態失敗");
			step := step + 10000;
		END_IF
		
	134:
		step := 140;
	
	140:
		IF GetEtherSta.devStates2[9].deviceState = 8 THEN
			step := step + 10;
		ELSE
			step := step + 1;
		END_IF
		
	141:
		GetEtherSta.ResetECat2(1010);
		step := step + 1;
		
	142:
		IF GetEtherSta.bBuzy OR GetEtherSta.bError THEN
			step := step + 1;
		END_IF
		
	143:
		IF GetEtherSta.bDone THEN
			step := step + 1;
		ELSIF GetEtherSta.bError THEN
			pMsg.Push_Alarm("重置Driver2-5 EtherCat狀態失敗");
			step := step + 10000;
		END_IF
		
	144:
		step := 150;
		
	150:
		IF GetEtherSta.devStates2[10].deviceState = 8 THEN
			step := step + 10;
		ELSE
			step := step + 1;
		END_IF
		
	151:
		GetEtherSta.ResetECat2(1011);
		step := step + 1;
		
	152:
		IF GetEtherSta.bBuzy OR GetEtherSta.bError THEN
			step := step + 1;
		END_IF
		
	153:
		IF GetEtherSta.bDone THEN
			step := step + 1;
		ELSIF GetEtherSta.bError THEN
			pMsg.Push_Alarm("重置Driver2-6 EtherCat狀態失敗");
			step := step + 10000;
		END_IF
		
	154:
		bDone := TRUE;
		step := 0;
END_CASE

METHOD Start : BOOL
VAR_INPUT
END_VAR
bDone := FALSE;
step := 1;
END_METHOD

END_PROGRAM

// ---- POUs/功能塊/EtherCat相關/GetEtherSta.TcPOU
PROGRAM GetEtherSta
VAR
	fbGetAllSlaveStates : FB_EcGetAllSlaveStates;
    sNetId      AT %I*  : AMSNETID ;
	sNetId2      AT %I*  : AMSNETID ;
    bExecute            : BOOL;
    devStates           : ARRAY[0..255] OF ST_EcSlaveState;
	devStates2           : ARRAY[0..255] OF ST_EcSlaveState;
    nSlaves             : UINT := 0;
	nSlaves2             : UINT := 0;
    nErrId              : UDINT;
	
	fbEcReqSlaveState : FB_EcReqSlaveState;
	
	fb_EcGetSlaveTopologyInfo	: FB_EcGetSlaveTopologyInfo;
	TopologyInfo 				: ARRAY[0..255] OF ST_TopologyDataEx;
	
	step: INT;
	tmr1: TON;
	i: UINT;
	
	fb_EcSetSlaveState : FB_EcSetSlaveState;
	resetSlaveNumber : INT;
	tmr100: TON;
	str_TmpString: WSTRING;
	
	
	
	step100: INT;
END_VAR

VAR_OUTPUT
	bErrorGetEC: BOOL;

	bBuzy: BOOL;
	bError: BOOL;
	bDone: BOOL;
	iErrorId : INT;
END_VAR

fbGetAllSlaveStates();
bErrorGetEC := fbGetAllSlaveStates.bError;
nErrId := fbGetAllSlaveStates.nErrId;

CASE step OF
	0:
		fb_EcGetSlaveTopologyInfo.sNetId	:= F_CreateAmsNetId(sNetId);
		fb_EcGetSlaveTopologyInfo.pAddrBuf	:= ADR(TopologyInfo);
		fb_EcGetSlaveTopologyInfo.cbBufLen	:= SIZEOF(TopologyInfo);
		fb_EcGetSlaveTopologyInfo.bExecute	:= TRUE;
		step := step + 1;
		
	1:
		IF fb_EcGetSlaveTopologyInfo.bBusy OR fb_EcGetSlaveTopologyInfo.bError THEN
			step := step + 1;
		END_IF
		
	2:
		IF NOT fb_EcGetSlaveTopologyInfo.bBusy THEN
			fb_EcGetSlaveTopologyInfo.bExecute := FALSE;
			step := step + 1;
		END_IF
		
	3:
		step := 10;
		
		
	10:
		fbGetAllSlaveStates.sNetId:= F_CreateAmsNetId(sNetId);
		fbGetAllSlaveStates.pStateBuf	:= ADR(devStates);
		fbGetAllSlaveStates.cbBufLen	:= SIZEOF(devStates);
		fbGetAllSlaveStates.bExecute := TRUE;
		step := step + 1;
		
	11:
		IF fbGetAllSlaveStates.bBusy OR fbGetAllSlaveStates.bError THEN
			step := step + 1;
		END_IF
		
	12:
		IF NOT fbGetAllSlaveStates.bBusy THEN
			fbGetAllSlaveStates.bExecute := FALSE;
			nSlaves := fbGetAllSlaveStates.nSlaves;
			step := step + 1;
		END_IF
		
	13:
		fbGetAllSlaveStates.sNetId		:= F_CreateAmsNetId(sNetId2);
		fbGetAllSlaveStates.pStateBuf	:= ADR(devStates2);
		fbGetAllSlaveStates.cbBufLen	:= SIZEOF(devStates2);
		fbGetAllSlaveStates.bExecute := TRUE;
		step := step + 1;
		
	14:
		IF fbGetAllSlaveStates.bBusy OR fbGetAllSlaveStates.bError THEN
			step := step + 1;
		END_IF
		
	15:
		IF NOT fbGetAllSlaveStates.bBusy THEN
			fbGetAllSlaveStates.bExecute := FALSE;
			nSlaves2 := fbGetAllSlaveStates.nSlaves;
			step := step + 1;
		END_IF
		
	16:
		FOR i := 0 TO nSlaves2 DO
			devStates[nSlaves + i] := devStates2[i];
		END_FOR
		step := 20;
		
		
	20:
		tmr1.in := TRUE;
		tmr1.pt := T#5S;
		IF tmr1.Q THEN
			tmr1.in := FALSE;
			step := step + 1;
		END_IF
		
	21:
		step := 10;
			
		
END_CASE

fb_EcGetSlaveTopologyInfo();

fbEcReqSlaveState();

Step100_resetECAT();

tmr1();

METHOD ResetECat1 : BOOL
VAR_INPUT
	SlaveAddr : INT;
	
END_VAR
resetSlaveNumber := SlaveAddr;
fb_EcSetSlaveState.sNetId := F_CreateAmsNetId(sNetId);
bDone := FALSE;
step100 := 100;
END_METHOD

METHOD ResetECat2 : BOOL
VAR_INPUT
	SlaveAddr : INT;
	
END_VAR
resetSlaveNumber := SlaveAddr;
fb_EcSetSlaveState.sNetId := F_CreateAmsNetId(sNetId2);
bDone := FALSE;
step100 := 100;
END_METHOD

ACTION Step100_resetECAT:
bBuzy := step100 > 0 AND step100 < 10000;
bError := step100 > 10000;

IF (EStop OR SystemError) THEN
	bDone := FALSE;
	IF bBuzy THEN
		step100 := step100  + 10000;
	END_IF
END_IF

IF ProgramReset THEN
	iErrorId := step;
	step := 0;
END_IF

CASE step100 OF
	100:
		fb_EcSetSlaveState.bExecute := FALSE;
		fb_EcSetSlaveState.tTimeout := T#5S;
		step100 := step100 + 1;
		
	101:// 將裝置設定狀態設為init
		fb_EcSetSlaveState.nSlaveAddr := INT_TO_UINT(resetSlaveNumber);
		fb_EcSetSlaveState.reqState := 1;
		fb_EcSetSlaveState.bExecute := TRUE;
		step100 := step100 + 1;
		
		
	102:
		IF fb_EcSetSlaveState.bBusy OR fb_EcSetSlaveState.bError THEN
			step100 := step100 + 1;
		END_IF
		
	103:
		IF fb_EcSetSlaveState.currState.deviceState = 1 THEN
			fb_EcSetSlaveState.bExecute := FALSE;
			step100 := step100 + 1;
		ELSIF fb_EcSetSlaveState.bError THEN
			fb_EcSetSlaveState.bExecute := FALSE;
			str_TmpString := WCONCAT(STR1:= "設定EtherCat站號", STR2:= INT_TO_WSTRING(resetSlaveNumber));
			str_TmpString := WCONCAT(STR1:= str_TmpString, STR2:= " 的狀態為INIT時發生錯誤");
			pMsg.Push_Alarm(str_TmpString);
			step100 := step100 + 10000;
		END_IF
	
	104:
		tmr100.IN:=TRUE;
		tmr100.PT := T#500MS;
		IF tmr100.Q THEN
			tmr100.IN:=FALSE;
			step100 := step100 + 1;
		END_IF
		
	105:
		step100 := 110;
		
		
		
	110:// 將裝置設定狀態設為PREOP 
		fb_EcSetSlaveState.nSlaveAddr := INT_TO_UINT(resetSlaveNumber);
		fb_EcSetSlaveState.reqState := 2;
		fb_EcSetSlaveState.bExecute := TRUE;
		step100 := step100 + 1;
		
	111:
		IF fb_EcSetSlaveState.bBusy OR fb_EcSetSlaveState.bError THEN
			step100 := step100 + 1;
		END_IF
		
	112:
		IF fb_EcSetSlaveState.currState.deviceState = 2 THEN
			fb_EcSetSlaveState.bExecute := FALSE;
			step100 := step100 + 1;
		ELSIF fb_EcSetSlaveState.bError THEN
			fb_EcSetSlaveState.bExecute := FALSE;
			str_TmpString := WCONCAT(STR1:= "設定EtherCat站號", STR2:= INT_TO_WSTRING(resetSlaveNumber));
			str_TmpString := WCONCAT(STR1:= str_TmpString, STR2:= " 的狀態為PREOP時發生錯誤");
			pMsg.Push_Alarm(str_TmpString);
			step100 := step100 + 10000;
		END_IF
		
	113:
		tmr100.IN:=TRUE;
		tmr100.PT := T#500MS;
		IF tmr100.Q THEN
			tmr100.IN:=FALSE;
			step100 := step100 + 1;
		END_IF
		
	114:
		step100 := 120;
		
		
		
	120:// 將裝置設定狀態設為SAFEOP
		fb_EcSetSlaveState.nSlaveAddr := INT_TO_UINT(resetSlaveNumber);
		fb_EcSetSlaveState.reqState := 4;
		fb_EcSetSlaveState.bExecute := TRUE;
		step100 := step100 + 1;
		
		
	121:
		IF fb_EcSetSlaveState.bBusy OR fb_EcSetSlaveState.bError THEN
			step100 := step100 + 1;
		END_IF
		
	122:
		IF fb_EcSetSlaveState.currState.deviceState = 4 THEN
			fb_EcSetSlaveState.bExecute := FALSE;
			step100 := step100 + 1;
		ELSIF fb_EcSetSlaveState.bError THEN
			fb_EcSetSlaveState.bExecute := FALSE;
			str_TmpString := WCONCAT(STR1:= "設定EtherCat站號", STR2:= INT_TO_WSTRING(resetSlaveNumber));
			str_TmpString := WCONCAT(STR1:= str_TmpString, STR2:= " 的狀態為SAFEOP時發生錯誤");
			pMsg.Push_Alarm(str_TmpString);
			step100 := step100 + 10000;
		END_IF
		
	123:
		tmr100.IN:=TRUE;
		tmr100.PT := T#500MS;
		IF tmr100.Q THEN
			tmr100.IN:=FALSE;
			step100 := step100 + 1;
		END_IF
		
	124:
		step100 := 130;
		
	130:// 將裝置設定狀態設為OP
		fb_EcSetSlaveState.nSlaveAddr := INT_TO_UINT(resetSlaveNumber);
		fb_EcSetSlaveState.reqState := 8;
		fb_EcSetSlaveState.bExecute := TRUE;
		step100 := step100 + 1;
		
		
	131:
		IF fb_EcSetSlaveState.bBusy OR fb_EcSetSlaveState.bError THEN
			step100 := step100 + 1;
		END_IF
		
	132:
		IF fb_EcSetSlaveState.currState.deviceState = 8 THEN
			fb_EcSetSlaveState.bExecute := FALSE;
			step100 := step100 + 1;
		ELSIF fb_EcSetSlaveState.bError THEN
			fb_EcSetSlaveState.bExecute := FALSE;
			str_TmpString := WCONCAT(STR1:= "設定EtherCat站號", STR2:= INT_TO_WSTRING(resetSlaveNumber));
			str_TmpString := WCONCAT(STR1:= str_TmpString, STR2:= " 的狀態為SAFEOP時發生錯誤");
			pMsg.Push_Alarm(str_TmpString);
			step100 := step100 + 10000;
		END_IF
		
	133:
		tmr100.IN:=TRUE;
		tmr100.PT := T#500MS;
		IF tmr100.Q THEN
			tmr100.IN:=FALSE;
			step100 := step100 + 1;
		END_IF
		
	134:
		bDone := TRUE;
		step100 := 0;
		
END_CASE

tmr100();
fb_EcSetSlaveState();
END_ACTION

END_PROGRAM

// ---- POUs/功能塊/RW_Config.TcPOU
PROGRAM RW_Config
VAR
	File_Path: STRING(INT#80) := '\Hard Disk2\Config\';
	fb_recipemancommands:recipemancommands;
	result: ARRAY [0..6] OF DWORD;
	result1: BOOL;
	boot: BOOL := true;
	



	GetTime: FB_LocalSystemTime := (bEnable := TRUE);
	

	tmr2: TON;
	tmr3: TON;
	
	//	目前時間	
	TimeNow: DATE_AND_TIME;
	
	strTimeNow: STRING;
END_VAR

VAR_INPUT
	// 寫入檔案
	Wrtie: BOOL;
END_VAR

tmr2(in:=boot, PT:=T#5S);
tmr3(in:=result1, PT:=T#1S);
IF tmr2.Q THEN
	result1 := fb_recipemancommands.SetStoragePath(File_Path);
	IF  tmr3.Q THEN
//		result[0] := fb_recipemancommands.LoadAndWriteRecipe('Config','Diff');
//		IF result[0] <> 0 THEN
//			result[1] := fb_recipemancommands.LoadRecipe('Config','Diff');
//			result[2] := fb_recipemancommands.WriteRecipe('Config','Diff');
//		END_IF
//		result1 := FALSE;
		boot := FALSE;
		Wrtie := TRUE;
	END_IF
END_IF

IF Wrtie THEN
	result1 := fb_recipemancommands.SetStoragePath(File_Path);
	result[3] := fb_recipemancommands.ReadRecipe('Config', 'Diff');
	result[4] := fb_recipemancommands.SaveRecipe('Config', 'Diff');
	result[5] := fb_recipemancommands.ReadAndSaveAs('Config','Diff');
	result[6] := fb_recipemancommands.ReadAndSaveRecipeAs('Config', 'Diff', CONCAT(STR1:= 'config_', STR2:= strTimeNow));
	Wrtie := FALSE;
END_IF



GetTime();
TimeNow:=SYSTEMTIME_TO_DT(GetTime.systemTime);
strTimeNow := CONCAT(STR1:= WORD_TO_STRING(GetTime.systemTime.wYear), STR2:='_');
strTimeNow := CONCAT(strTimeNow ,CONCAT(STR1:= WORD_TO_STRING(GetTime.systemTime.wMonth), STR2:='_'));
strTimeNow := CONCAT(strTimeNow ,CONCAT(STR1:= WORD_TO_STRING(GetTime.systemTime.wDay), STR2:='_'));
strTimeNow := CONCAT(strTimeNow ,WORD_TO_STRING(GetTime.systemTime.wHour));

END_PROGRAM

// ---- POUs/功能塊/字串處理功能塊/字串填充/FILLSTRING.TcPOU
FUNCTION FILLSTRING : STRING
VAR_INPUT
	str : STRING;
	strlen : INT;
	fill_char : STRING(1);
END_VAR
VAR
	rawlen : INT;
	
	fillNumber : INT;
	
	tmpstr : STRING;
	
	i : INT;
END_VAR

rawlen := LEN(STR:= str);

fillNumber := strlen - rawlen;

tmpstr := '';

FOR i:= 1 TO fillNumber DO
	tmpstr := CONCAT(STR1:= tmpstr, STR2:= fill_char);
END_FOR

FILLSTRING := CONCAT(STR1:= tmpstr, STR2:= str);

END_FUNCTION

// ---- POUs/功能塊/字串處理功能塊/字串連接/StrConcat.TcPOU
FUNCTION StrConcat : STRING(511)
VAR_INPUT
	str0 : STRING(511) := '';
	str1 : STRING(511) := '';
	str2 : STRING(511) := '';
	str3 : STRING(511) := '';
	str4 : STRING(511) := '';
	str5 : STRING(511) := '';
	str6 : STRING(511) := '';
	str7 : STRING(511) := '';
	str8 : STRING(511) := '';
END_VAR
VAR
	tmpstr : STRING(511);
END_VAR

tmpstr := CONCAT(STR1:= str0, STR2:= str1);
tmpstr := CONCAT(STR1:= tmpstr, STR2:= str2);
tmpstr := CONCAT(STR1:= tmpstr, STR2:= str3);
tmpstr := CONCAT(STR1:= tmpstr, STR2:= str4);
tmpstr := CONCAT(STR1:= tmpstr, STR2:= str5);
tmpstr := CONCAT(STR1:= tmpstr, STR2:= str6);
tmpstr := CONCAT(STR1:= tmpstr, STR2:= str7);
tmpstr := CONCAT(STR1:= tmpstr, STR2:= str8);
StrConcat := tmpstr;
RETURN;

END_FUNCTION
